(* Timer *)
WaitValve		(IN:=  bValveTime, PT:=STRING_TO_TIME(CONCAT(tempTime, 'ms')), Q=>, ET=>); 		(*Timer*)		(* For waiting for Valves 				*)
Wait			(IN:=  bWait			, PT:=T#200MS, Q=>, ET=>); 		(*Timer*)		(* For testing 							*)
Wait2			(IN:=  bWait2			, PT:=T#2500MS, Q=>, ET=>);		(*Timer*)		(* For waiting for stem to stand still 	*)
WaitMotorDrive	(IN:=  bDriveTime		, PT:=T#500MS, Q=>, ET=>);		(*Timer*)		(* For Homing 							*)

(* uiStepsToMove			-->	Antal pulser på tællerkort	:	24 Pulser pr mm * antal mm 										*)
uiStepsToMove := INT_TO_UINT(24 * uiDistToGrab);

FB_OPEN_CUT		(ExecuteHmi := (sToolControl = 'cut-open') OR GbOpenCut, 	ControlType := 1,	Ack := uiSignalInToolAck.02, 	OutQ => uiSignalOutTool.02);
FB_CLOSE_CUT	(ExecuteHmi := (sToolControl = 'cut-close'),	ControlType := 1,	Ack := uiSignalInToolAck.03, 	OutQ => uiSignalOutTool.03);
FB_RELEASE_CUT	(ExecuteHmi := GbReleaseCut OR FB_RELEASE_CUT.Execute,	ControlType := 1,	Ack := uiSignalInToolAck.01, 	OutQ =>);
FB_OPEN_PICK	(ExecuteHmi := (sToolControl = 'pick-open') OR GbOpenPick,	ControlType := 1,	Ack := uiSignalInToolAck.04, 	OutQ => uiSignalOutTool.04);
FB_CLOSE_PICK	(ExecuteHmi := (sToolControl = 'pick-close'),	ControlType := 1,	Ack := uiSignalInToolAck.05, 	OutQ => uiSignalOutTool.05);

FB_LOAD_CUT		(ExecuteHmi := (sToolControl = 'cut-load'),		ControlType := 5, 	Ack := uiSignalInToolAck.00,	OutQ => uiSignalOutTool.00, 	OutQ2 => qValve1, 	OutQ3 => qValve2);
FB_DELOAD_CUT	(ExecuteHmi := (sToolControl = 'cut-deload') OR GbDeloadCut,	ControlType := 2, 	Ack := uiSignalInToolAck.01,	OutQ => , 	OutQ2 =>bValve1Control);

FB_OPEN_GRIP	(ExecuteHmi := (sToolControl = 'grip-open'),	ControlType := 4,	OutQ =>,);
FB_CLOSE_GRIP	(ExecuteHmi := (sToolControl = 'grip-close'),	ControlType := 3, 	OutQ => ,);

FB_BRAKE		(ControlType := 1, Ack := NOT FB_BRAKE.Execute, 	OutQ => qValve3);

IF (FB_RELEASE_CUT.Execute AND FB_RELEASE_CUT.State = 10) OR (FB_DELOAD_CUT.State = 110) THEN
	uiSignalOutTool.01 := TRUE;
ELSE
	uiSignalOutTool.01 := FALSE;
END_IF

IF (sToolControl = 'brake-activate') THEN
	FB_BRAKE.Execute := TRUE;
ELSIF (sToolControl = 'brake-deactivate') THEN
	FB_BRAKE.Execute := FALSE;
END_IF


IF GbCloseGrip OR FB_CLOSE_GRIP.Execute OR FB_CLOSE_GRIP.ExecuteHmi THEN
	FB_OPEN_GRIP.Execute := FALSE;
	qValve4 := FB_CLOSE_GRIP.OutQ;
	testing := FALSE;
END_IF
IF GbOpenGrip OR FB_OPEN_GRIP.Execute OR FB_OPEN_GRIP.ExecuteHmi THEN
	testing := TRUE;
	FB_CLOSE_GRIP.Execute := FALSE;
	qValve4 := NOT FB_OPEN_GRIP.OutQ;
END_IF


IF bValve1Control THEN
	qValve1 := TRUE;
END_IF

IF sToolControl = 'cut-close' THEN
	GbCloseCut := TRUE;
	
ELSE 
	GbCloseCut := FALSE;
END_IF

END_PROGRAM

// ---- POUs/CONTROLs/Control.TcPOU
PROGRAM Control
VAR_INPUT
	State: INT := 0;
	NewState: INT := 0;

	InternalState: INT := 0;
	InternalNewState: INT := 0;
END_VAR

VAR
	adsTest: INT;
	(* FUNCTION BLOCKS *)

	(* REALS *)
		
	(* INTEGERS *)
	(*uiTrunkPos: 		UINT;				(* Stamme position	-->	Afstand i mm.															*)
	iBunchPosZ: 		UINT;
	iStemAngle:		INT;

	uiCutCoordX: 		UINT;
	uiCutCoordY: 		UINT;
	uiCutCoordZ: 		UINT;

	iStemPosX: 		UINT;				(* *)
	iStemPosY: 		UINT;				(* *)
	iStemPosZ: 		UINT;
	iRoll: 			INT;
	iPitch: 			UINT;
	iYaw:			INT;
	iPickAngle: 		INT;*)

	ImageRetryHeight:	INT;

	iMoved: 			INT;					(* Hvor mange gange har cut bevæget sig efter iBunchPosZ er nået *)
	iCnfgChange:		INT := 0;
	uiDeleaf: 		UINT;

	(* BOOLS *)
	bStopped: BOOL;
	bRobotFail: BOOL;

	bRetry: INT;
	bStemGrabbed: BOOL;

	cartMoved: BOOL;
	cartX: USINT;
	testbreak: BOOL;
	distCutJoint: INT;
	cutMin: INT;
	testFail: BOOL;
	break: BOOL;
END_VAR

CASE State OF

	0: (* init - Every important variables will be resat before the start of the sequence *)
		IF bStart AND uiprogNo = 6 AND State <> 2000  AND NOT bAlarmState THEN
			uiStatus := 1;
			FB_BRAKE.Execute := TRUE;

			(* Init variables *)
			bRetry := 0;
			uiCalibImgCount	:= 0;
			iMoved := 0;
			iImageZone := 0;
			gJointFound := 0;
			gResetPcCom 	:= TRUE;
			iCnfgChange := 0;
			uiDeleaf := 0;
			bPosSentToPcCom := FALSE;
			gStopped := FALSE;

			(* Before starting - Home *)
			GbHomeGripStem := TRUE;
			IF bHomeDone THEN
				bStart := FALSE;
				bHomeDone := FALSE;
				NewState := 10;
			END_IF
		END_IF

	10:	(* Set velocity - Both Cut and Pick *)
		bLog := TRUE;	// Starts logging of data in this Control sequence
	
		FB_SET_VELOCITY.Execute := TRUE;
		uiSignalOutSpeedControl := PROGRAM_DATA.usiVelocity;
		uiSignalOutControl := FB_SET_VELOCITY.OutQ;
		IF FB_SET_VELOCITY.Done THEN
			FB_SET_VELOCITY.Execute := FALSE;
			NewState := 20;
		END_IF

	20:	(* Idle - Both Cut and Pick *)
		FB_MOVE_TO_IDLE.Execute := TRUE;
		uiSignalOutControl := FB_MOVE_TO_IDLE.OutQ;
		IF FB_MOVE_TO_IDLE.Done THEN
			FB_MOVE_TO_IDLE.Execute := FALSE;
			NewState := 30;
		END_IF




		(* ------------------------------------------------------------------- Get Stem  ------------------------------------------------------------------- *)
	30:	(*  Load cutter *)
		FB_LOAD_CUT.Execute := TRUE;
		IF FB_LOAD_CUT.Done THEN
			FB_LOAD_CUT.Execute := FALSE;
			NewState := 35;
		END_IF
		
	35:
		(* Close grip - for it not to be in the images from CutCam *)
		FB_CLOSE_GRIP.Execute := TRUE;
		IF FB_CLOSE_GRIP.Done THEN
			FB_CLOSE_GRIP.Execute := FALSE;
			NewState := 40;
		END_IF

	40: (* Cam 1 Take image	-	parameters recieved from Vision = height of lowest ripe tomato and Y coord for lowest point of the stem *)

		FB_CAM_ONE_CONTROL.Execute := TRUE;
		IF FB_CAM_ONE_CONTROL.Done THEN
			FB_CAM_ONE_CONTROL.Execute := FALSE;
			IF FB_CAM_ONE_CONTROL.Fail THEN
				(* Adjust cart height  in order to retry *)
				NewState := 1000;
			ELSE
				(* uiDistToGrab 	-->		Distance from Joris Gripper to stem 			*)
				uiDistToGrab	:= FB_CAM_ONE_CONTROL.TrunkDist;
				(* iBunchPosZ	-->		Height of the lowest hanging red tomato		*)
				iBunchPosZ 	:= FB_CAM_ONE_CONTROL.BunchHeight;
				(* i StemAngle	-->		Heading direction from stem to lowest tomato	*)
				iStemAngle	:= FB_CAM_ONE_CONTROL.StemHeading;
				(* iImageZone	-->		Zone of lowest tomato						*)
				iImageZone	:= FB_CAM_ONE_CONTROL.Zone;
				usiImageLog := usiImageLog + 1;
				NewState := 45;
			END_IF
		END_IF

	45: (* Open gripper after  *)
		IF bRetry < 3 THEN
			FB_OPEN_GRIP.Execute := TRUE;
			IF FB_OPEN_GRIP.Done THEN
				bRetry := bRetry + 1;
				usiRetryLog := usiRetryLog + 1;
				FB_OPEN_GRIP.Execute := FALSE;
				NewState := 50;
			END_IF
		ELSE
			NewState := 1000;
		END_IF


	50:				(* Joris gripper retreives stem *)
		(* Grab stem and pull in *)
		IF NOT bAck THEN
			(* HMI knap der kalder GribStem *)
			GbGripStem := TRUE;
		ELSIF bAck THEN
			gResetPcCom := TRUE;
			NewState := 55;
		END_IF

	55:
		(* Check if stem is grabed *)
		IF uiToolState = 0 THEN
			(* Retry to grab the stem with a larger uiDistToGrab *)
			IF bJorisSensor THEN
				CASE bRetry OF
					0:
						// Retry 50mm further aways
						uiDistToGrab := uiDistToGrab + 50;
						NewState := 45;
						
					1:
						// Why?
						uiDistToGrab := uiDistToGrab - 50;
						NewState := 60;
						
					2:
						(* Keep trying intil the stem is grabed *)
						bRetry := 0;
						
				ELSE
					NewState := 1000;
				END_CASE
			ELSE
				bRetry := 0;
				NewState := 100;
			END_IF
		END_IF
		
	60:
		(* Move cart so that the *)
		IF FB_CAM_ONE_CONTROL.TrunkPosX > 280 THEN
			(* Move cart forward *)
			(* Move cart FB_CAM_ONE_CONTROL.TrunkPosX - 280 *)
			cartMoved := TRUE;
		ELSE
			(* Move cart backward *)
			(* Move cart 280 - FB_CAM_ONE_CONTROL.TrunkPosX *)
			cartMoved := TRUE;
		END_IF
		NewState := 70;
	
	70:
		IF cartMoved THEN
			(* Take a new photo and retry *)
			IF bRetry < 2 THEN
				cartMoved := FALSE;
				usiRetryLog := usiRetryLog + 1;
				NewState := 40;
			ELSE
				cartMoved := FALSE;
				NewState := 45;
			END_IF
		END_IF














	(* ------------------------------------------------------------------- Grab Stem  ------------------------------------------------------------------- *)
	100:		(* Robot Pick move to Image Pos *)
		
		IF (ABS(iStemAngle) >= 90) THEN
			IF iStemAngle < 0 THEN
				gTomatoHeading := INT_TO_BYTE(270 - ABS(iStemAngle));
			ELSE
				gTomatoHeading := INT_TO_BYTE(ABS(iStemAngle) - 90);
			END_IF
		ELSE
			gTomatoHeading := 0;
		END_IF
		
		(*IF iStemAngle < 0 THEN
			gTomatoHeading := INT_TO_BYTE(ABS(iStemAngle));
		ELSE
			gTomatoHeading := 0;
		END_IF*)
		
		FB_PICK_TRUNK_IMAGE.Execute := TRUE;
		uiSignalOutControl := FB_PICK_TRUNK_IMAGE.OutQ;
		IF FB_PICK_TRUNK_IMAGE.Done THEN
			IF uiSignalInRobotFail.00 AND testFail THEN		// Hvad er testFail?
				NewState := 1000;
				bBackToZero := TRUE;
			ELSE
				FB_PICK_TRUNK_IMAGE.Execute := FALSE;
				gResetPcCom := TRUE;
				NewState := 110;
			END_IF
		END_IF

	110:		(* Send Robot Pick Position *)
		getPickCoords := TRUE;
		IF bPosSentToPcCom AND FB_GET_PICK_COORD.Execute = FALSE THEN
			ImageRetryHeight := stDataToVision.CoordZR2G;
			bPosSentToPcCom := FALSE;
			bGetCoordDone := FALSE;
			NewState := 120;
		END_IF

	120:		(* Cam 2 take image *)
		(* Take bottom Image *)
		(* If pick coordinates are recieved, take an image *)
		IF stDataToVision.CoordXR2G <> 0 AND stDataToVision.CoordYR2G <> 0 AND stDataToVision.CoordZR2G <> 0 THEN
			FB_CAM_TWO_CONTROL.Execute := TRUE;
			IF FB_CAM_TWO_CONTROL.Done THEN
				(* If the positions was unacceptable  - Prepare to take a new picture from 50 mm further up *)
				IF FB_CAM_TWO_CONTROL.Fail THEN
					(* Send new pos to Robots *)
					GviX	:= stDataToVision.CoordXR2G / 10;
					GviY 	:= stDataToVision.CoordYR2G / 10;
					GviZ 	:= (stDataToVision.CoordZR2G / 10) + 50;

					(* GsendCoord			-->	Starter SendCoordinates sekvensen							-	Sender koordinater til robotterne 		*)
					(* uiSignalOutShared.06	-->	Bekræftelse på at koordinaterne er sendt til udgangene i box 10	-	Acknowledge fra SendCoordinates	*)
					GsendCoord := TRUE;
					IF uiSignalOutShared.06 THEN
						(* Send_pos	-->	Kommando der fortæller robot cut at nogle nye positioner er sendt *)
						uiSignalOutControl := Send_pos;
					END_IF
					IF uiSignalInAck = Send_pos THEN
						FB_CAM_TWO_CONTROL.Execute := FALSE;
						uiSignalOutControl := 0;
						uiCalibImgCount := uiCalibImgCount + 1;
						usiImageLog := usiImageLog + 1;
						NewState := 130;
					END_IF
				ELSE
					(* If positions are acceptable and stem is found, Send the posiotions to the robots *)
					FB_CAM_TWO_CONTROL.Execute := FALSE;
					IF stDataFromVision.gStemFound = 1 THEN
						IF (FB_CAM_TWO_CONTROL.X < 400) AND (FB_CAM_TWO_CONTROL.Y < 450) AND (FB_CAM_TWO_CONTROL.Z < 1000) and (FB_CAM_TWO_CONTROL.X > 0) AND (FB_CAM_TWO_CONTROL.Y > 150) AND (FB_CAM_TWO_CONTROL.Z > 200) THEN
							GviX	:= FB_CAM_TWO_CONTROL.X;
							GviY 	:= FB_CAM_TWO_CONTROL.Y;
							//Hvis joint fundet, tag fat 10cm længere nede.
							IF stDataFromVision.gJointFound = 1 THEN
								GviZ 	:= FB_CAM_TWO_CONTROL.Z - 100;
							ELSE
								GviZ 	:= FB_CAM_TWO_CONTROL.Z;
							END_IF
							//Tjek om klasen hænger i vejen for CutTool. Hvis ja, tag fat længere nede.
							IF iStemAngle < -75 AND iStemAngle > -105 AND FB_CAM_TWO_CONTROL.Z > iBunchPosZ THEN
								GviZ := iBunchPosZ;
							END_IF
							IF GviZ < 200 THEN
								GviZ := 200;
							END_IF
							GviA 	:= FB_CAM_TWO_CONTROL.RotZ0;
							GviE 	:= FB_CAM_TWO_CONTROL.RotY;
							GviR 	:= FB_CAM_TWO_CONTROL.RotZ1;
	
							GviX2 	:= FB_CAM_TWO_CONTROL.X;
							GviY2 	:= (FB_CAM_TWO_CONTROL.Y + FB_CAM_TWO_CONTROL.Y + FB_CAM_ONE_CONTROL.Y)/3;
							GviZ2	:= GviZ;
							(*GviZ2 	:= FB_CAM_ONE_CONTROL.Z + 50;*)
	
							iImageZone	:= FB_CAM_ONE_CONTROL.Zone;
							usiImageLog := usiImageLog + 1;
							NewState := 150;
						END_IF
					(* IF the stem cannot be found, retry grabbing the stem with Joris gripper *)
					ELSE
						IF bRetry = 0 THEN
							bRetry := 1;
							usiRetryLog := usiRetryLog + 1;
							gResetPcCom := TRUE;
							NewState := 110;
						ELSE
							gResetPcCom := TRUE;
							bRetry := 1000;
							bBackToZero := TRUE;
						END_IF
					END_IF
				END_IF
			END_IF
		END_IF


	130:
		IF uiSignalInAck = 0 THEN
			IF bRetry = 0 THEN
				bRetry := bRetry + 1;
				usiRetryLog := usiRetryLog + 1;
				NewState := 100;
			ELSE
				bRetry := 1000;
				bBackToZero := TRUE;
			END_IF
		END_IF

	150:		(* Send Pos to Robot *)

		(* GsendCoord			-->	Starter SendCoordinates sekvensen							-	Sender koordinater til robotterne 		*)
		(* uiSignalOutShared.06	-->	Bekræftelse på at koordinaterne er sendt til udgangene i box 10	-	Acknowledge fra SendCoordinates	*)
		GsendCoord := TRUE;
		IF uiSignalOutShared.06 THEN
			(* Send_pos	-->	Kommando der fortæller robot cut at nogle nye positioner er sendt *)
			uiSignalOutControl := Send_two_pos;
		END_IF

		IF uiSignalInAck = Send_two_pos THEN
			uiSignalOutControl := 0;
			uiCalibImgCount := uiCalibImgCount + 1;
			NewState := 155;
		END_IF


	155:
		IF uiSignalInAck = 0 THEN
			NewState := 160;
		END_IF

	160:		(* Grab the stem + Move to image pos *)
		FB_IMAGE_GRAB.Execute := TRUE;
		uiSignalOutControl := FB_IMAGE_GRAB.OutQ;

		IF FB_IMAGE_GRAB.Done THEN
			IF uiSignalInRobotFail.00 AND testFail THEN
				NewState := 1000;
				bBackToZero := TRUE;
			ELSE
				FB_IMAGE_GRAB.Execute := FALSE;
				NewState := 200;
			END_IF
		END_IF









	(* ------------------------------------------------------------------- "WHAT IF" FIXES  ------------------------------------------------------------------- *)
	200:
		IF NOT bRobotFail THEN
			bRetry := 0;
			gResetPcCom := TRUE;
			NewState := 250;
		ELSE
			(* Retries:																						*)
			(* Open and close cone								-	To check if it was a misreading from sensor 	*)
			(* Move to pos 50mm above normal image pos, then retry												*)
			IF bRetry  < 2 THEN
				bRetry := bRetry + 1;
				usiRetryLog := usiRetryLog + 1;
				(*uiCalibImgCount := 0;*)
				GviZ2 := stDataToVision.CoordZR2G/10 + 100;
				NewState := 220;
			ELSE
				bBackToZero := TRUE;
			END_IF
		END_IF


	220:
		(* GsendCoord			-->	Starter SendCoordinates sekvensen							-	Sender koordinater til robotterne 		*)
		(* uiSignalOutShared.06	-->	Bekræftelse på at koordinaterne er sendt til udgangene i box 10	-	Acknowledge fra SendCoordinates	*)
		GsendCoord := TRUE;
		IF uiSignalOutShared.06 THEN
			(* Send_pos	-->	Kommando der fortæller robot cut at nogle nye positioner er sendt *)
			uiSignalOutControl := Send_two_pos;
		END_IF

		IF uiSignalInAck = Send_two_pos THEN
			uiSignalOutControl := 0;
			NewState := 225;
		END_IF

	225:
		IF uiSignalInAck = 0 THEN
			gResetPcCom := TRUE;
			NewState := 230;
		END_IF


	230:		(* Retry Grab Stem *)
		FB_RETRY_GRAB_STEM.Execute := TRUE;
		uiSignalOutControl := FB_RETRY_GRAB_STEM.OutQ;
		IF FB_RETRY_GRAB_STEM.Done THEN
			FB_RETRY_GRAB_STEM.Execute := FALSE;
			gResetPcCom := TRUE;
			NewState := 110;
		END_IF










	(* ------------------------------------------------------------------- Move On Stem  ------------------------------------------------------------------- *)
	250:		(* Send Robot Pick Position *)
		getPickCoords := TRUE;
		IF bPosSentToPcCom AND FB_GET_PICK_COORD.Execute = FALSE THEN
			ImageRetryHeight := stDataToVision.CoordZR2G;
			bPosSentToPcCom := FALSE;
			bGetCoordDone := FALSE;
			NewState := 260;
		END_IF

	260:
		IF stDataToVision.CoordXR2G <> 0 AND stDataToVision.CoordYR2G <> 0 AND stDataToVision.CoordZR2G <> 0 THEN
			FB_CAM_TWO_CONTROL.Execute := TRUE;
			IF FB_CAM_TWO_CONTROL.Done THEN
				FB_CAM_TWO_CONTROL.Execute := FALSE;
				(* Check if the stem is found *)
				IF FB_CAM_TWO_CONTROL.StemFound = 1 THEN
					IF FB_CAM_TWO_CONTROL.X > 350 OR FB_CAM_TWO_CONTROL.X < 200 OR FB_CAM_TWO_CONTROL.Y > 350 OR FB_CAM_TWO_CONTROL.Y < 200 THEN
						GviX := 320;
						GviY := 320;
						IF (stDataFromVision.ResultPar3 < iBunchPosZ) THEN
							GviZ := FB_CAM_TWO_CONTROL.Z;
						ELSE
							GviZ := iBunchPosZ;
						END_IF
						GviA := 0;
						GviE := 0;
						GviR := 40;
					ELSE
						GviX := (FB_CAM_TWO_CONTROL.X + 320) / 2;
						GviY := (FB_CAM_TWO_CONTROL.Y + 320) / 2;
						IF (stDataFromVision.ResultPar3 < iBunchPosZ) THEN
							GviZ := FB_CAM_TWO_CONTROL.Z;
						ELSE
							GviZ := iBunchPosZ;
						END_IF
						GviA := 0;
						GviE := 0;
						GviR := 40;
					END_IF
					(*IF FB_CAM_TWO_CONTROL.JointFound = 1 THEN
						GviPick := FB_CAM_TWO_CONTROL.PickAngle;
						iImageZone := FB_CAM_TWO_CONTROL.Zone;
						gResetPcCom := TRUE;
						NewState := 310;
					ELSE*)
					usiImageLog := usiImageLog + 1;
						gResetPcCom := TRUE;
						NewState := 270;
					(*END_IF*)
				ELSE
					usiImageLog := usiImageLog + 1;
					gResetPcCom := TRUE;
					NewState := 345;
				END_IF
			END_IF
		END_IF

	270:
		(* Send pos to Robots *)
		(* GsendCoord			-->	Starter SendCoordinates sekvensen							-	Sender koordinater til robotterne 		*)
		(* uiSignalOutShared.06	-->	Bekræftelse på at koordinaterne er sendt til udgangene i box 10	-	Acknowledge fra SendCoordinates	*)
		GsendCoord := TRUE;
		IF uiSignalOutShared.06 THEN
			(* Send_pos	-->	Kommando der fortæller robot cut at nogle nye positioner er sendt *)
			uiSignalOutControl := Send_pos;
		END_IF
		IF uiSignalInAck = Send_pos THEN
			uiSignalOutControl := 0;
			uiCalibImgCount := uiCalibImgCount + 1;
			NewState := 275;
		END_IF

	275:
		IF uiSignalInAck = 0 THEN
			NewState := 280;
		END_IF

	280:		(* CO-MOVE up the stem *)
		FB_COMOVE_IMAGE.Execute := TRUE;
		uiSignalOutControl := FB_COMOVE_IMAGE.OutQ;
		IF FB_COMOVE_IMAGE.Done THEN
			IF uiSignalInRobotFail.00 AND testFail THEN
				NewState := 1000;
				bBackToZero := TRUE;
			ELSE
				FB_COMOVE_IMAGE.Execute := FALSE;
				IF bRobotFail THEN
					NewState := 3000;
				ELSE
					NewState := 290;
				END_IF
			END_IF
		END_IF

	290:
		(* Send Pick coordinate *)
		(* Send Pick pos to PcCom for next image *)
		getPickCoords := TRUE;
		IF bPosSentToPcCom AND FB_GET_PICK_COORD.Execute = FALSE THEN
			bPosSentToPcCom := FALSE;
			NewState := 300;
		END_IF











	(* ------------------------------------------------------------------- Find Joint  ------------------------------------------------------------------- *)
	300:		(* Take a picture *)
		IF stDataToVision.CoordXR2G <> 0 AND stDataToVision.CoordYR2G <> 0 AND stDataToVision.CoordZR2G <> 0 THEN
			FB_CAM_TWO_CONTROL.Execute := TRUE;
			IF FB_CAM_TWO_CONTROL.Done THEN
				IF FB_CAM_TWO_CONTROL.StemFound = 1 THEN
					IF FB_GET_CUT_COORD.Execute = FALSE THEN
						IF FB_CAM_TWO_CONTROL.Zone <> 0 THEN
							iImageZone := FB_CAM_TWO_CONTROL.Zone;
						END_IF
						IF distCutJoint = 0 THEN
							(* Get Cut coord *)
							gResetPcCom := TRUE;
							getCutCoords := TRUE;
							bGetCutCoordDone:= FALSE;
							cutMin := 15;	(* Max lenght from top of cut head to joint*)
						END_IF
						IF FB_CAM_TWO_CONTROL.X > 350 OR FB_CAM_TWO_CONTROL.X < 200 OR FB_CAM_TWO_CONTROL.Y > 350 OR FB_CAM_TWO_CONTROL.Y < 200 THEN
							usiImageLog := usiImageLog + 1;
							NewState := 302;							
						ELSE
							usiImageLog := usiImageLog + 1;
							NewState := 303;
						END_IF
					END_IF
				ELSE
					FB_CAM_TWO_CONTROL.Execute := FALSE;
					gResetPcCom := TRUE;
					usiImageLog := usiImageLog + 1;
					NewState := 345;
				END_IF
			END_IF
		END_IF
		
	302:
		IF bGetCutCoordDone THEN
			bGetCutCoordDone:= FALSE;
			distCutJoint := stDataFromVision.ResultPar3 - (currentRobotZ / 10);
		
			IF distCutJoint <> 0 OR ((stDataFromVision.ResultPar3 = (currentRobotZ/10)) AND (currentRobotZ <> 0)) THEN
				IF FB_CAM_TWO_CONTROL.JointFound = 1 AND distCutJoint <= cutMin THEN
					GviPick := FB_CAM_TWO_CONTROL.PickAngle;

					getCutCoords := TRUE;
					IF FB_CAM_TWO_CONTROL.TrussFound = 1 THEN
						iCnfgChange := 0;
					END_IF
					IF bPosSentToPcCom AND FB_GET_CUT_COORD.Execute = FALSE THEN
						bPosSentToPcCom := FALSE;
						FB_CAM_TWO_CONTROL.Execute := FALSE;
						gResetPcCom := TRUE;
						NewState := 305;
					END_IF
				ELSE
					GviX := 320;
					GviY := 320;
					GviZ := FB_CAM_TWO_CONTROL.Z;

					GviA 	:= 0;
					GviE 	:= 0;
					GviR 	:= 40;

					FB_CAM_TWO_CONTROL.Execute := FALSE;
					gResetPcCom := TRUE;
					iCnfgChange := 0;
					NewState := 310;
				END_IF
			END_IF
		END_IF
		
	303:
		IF bGetCutCoordDone THEN
			bGetCutCoordDone:= FALSE;
			distCutJoint := stDataFromVision.ResultPar3 - (currentRobotZ / 10);
		
			IF distCutJoint <> 0 OR ((stDataFromVision.ResultPar3 = (currentRobotZ/10)) AND (currentRobotZ <> 0)) THEN
				IF FB_CAM_TWO_CONTROL.JointFound = 1 AND distCutJoint <= cutMin THEN
					GviPick := FB_CAM_TWO_CONTROL.PickAngle;
					IF FB_CAM_TWO_CONTROL.TrussFound = 1 THEN
						iCnfgChange := 0;
					END_IF
					IF bPosSentToPcCom THEN
						bPosSentToPcCom := FALSE;
						FB_CAM_TWO_CONTROL.Execute := FALSE;
						NewState := 305;
					END_IF
				ELSIF distCutJoint > cutMin THEN
					IF FB_CAM_TWO_CONTROL.JointFound = 1 THEN
						GviZ := FB_CAM_TWO_CONTROL.Z - 10;
						iCnfgChange := 0;
					ELSE
						GviZ := FB_CAM_TWO_CONTROL.Z;
					END_IF
					GviX := (FB_CAM_TWO_CONTROL.X + 320) / 2;
					GviY := (FB_CAM_TWO_CONTROL.Y + 320) / 2;
					GviA 	:= 0;
					GviE 	:= 0;
					GviR 	:= 40;

					FB_CAM_TWO_CONTROL.Execute := FALSE;
					gResetPcCom := TRUE;
					NewState := 310;
				ELSE
					bBackToZero := TRUE;
				END_IF
			END_IF
		END_IF

	305:
		IF uiSignalInAck = 0 THEN
			GviX	:= stDataToVision.CoordXR1G / 10;
			GviY	:= stDataToVision.CoordYR1G / 10;
			GviZ	:= stDataToVision.CoordZR1G / 10;
			gResetPcCom := TRUE;
			NewState := 310;
		END_IF

	310:		(* Send pos *)
		(* GsendCoord			-->	Starter SendCoordinates sekvensen							-	Sender koordinater til robotterne 		*)
		(* uiSignalOutShared.06	-->	Bekræftelse på at koordinaterne er sendt til udgangene i box 10	-	Acknowledge fra SendCoordinates	*)
		IF (FB_CAM_TWO_CONTROL.TomatoFound = 1) AND (FB_CAM_TWO_CONTROL.JointFound <> 1) THEN
			NewState := 315;
		ELSE
			GsendCoord := TRUE;
			IF uiSignalOutShared.06 THEN
				(* Send_pos	-->	Kommando der fortæller robot cut at nogle nye positioner er sendt *)
				uiSignalOutControl := Send_pos;
			END_IF
			IF uiSignalInAck = Send_pos THEN
				uiSignalOutControl := 0;
				(*uiCalibImgCount := uiCalibImgCount + 1;*)
				NewState := 315;
			END_IF
		END_IF

	315:
		IF uiSignalInAck = 0 THEN
			IF FB_CAM_TWO_CONTROL.JointFound = 1 AND stDataFromVision.ResultPar3 > iBunchPosZ AND (currentRobotZ/10) > iBunchPosZ AND distCutJoint < cutMin THEN
				NewState := 345;
			ELSIF (FB_CAM_TWO_CONTROL.TomatoFound = 1) AND (FB_CAM_TWO_CONTROL.JointFound <> 1) AND (stDataFromVision.ResultPar3 > iBunchPosZ) AND iCnfgChange < 6 THEN
				iCnfgChange := iCnfgChange + 1;
				usiImageRetry := usiImageRetry + 1;
				IF uiCalibImgCount < 50 THEN
					uiCalibImgCount := 50;
				END_IF
				IF uiCalibImgCount >= 50 AND uiCalibImgCount <= 200 THEN
					NewState := 350;
				ELSIF uiCalibImgCount = 250 THEN
					NewState := 450;
				END_IF
			ELSE
				NewState := 320;
			END_IF
		END_IF
	320:
		FB_COMOVE_IMAGE.Execute := TRUE;
		uiSignalOutControl := FB_COMOVE_IMAGE.OutQ;
		IF FB_COMOVE_IMAGE.Done THEN
			FB_COMOVE_IMAGE.Execute := FALSE;
			IF uiSignalInRobotFail.00 AND testFail THEN
				NewState := 1000;
				bBackToZero := TRUE;
			ELSE
				IF bRobotFail THEN
					NewState := 3000;
				ELSE
					IF FB_CAM_TWO_CONTROL.JointFound = 1 AND distCutJoint > cutMin AND stDataFromVision.ResultPar3 < iBunchPosZ AND FB_CAM_TWO_CONTROL.TrussFound = 0 THEN
						NewState := 325;
					ELSE
						NewState := 330;
					END_IF
				END_IF
			END_IF
		END_IF

	325:
		FB_RELEASE_CUT.Execute := TRUE;
		IF FB_RELEASE_CUT.Done THEN
			usiStickoutCutLog := usiStickoutCutLog + 1;
			FB_RELEASE_CUT.Execute := FALSE;
			NewState := 327;
		END_IF

	327:
		FB_LOAD_CUT.Execute := TRUE;
		IF FB_LOAD_CUT.Done THEN
			FB_LOAD_CUT.Execute := FALSE;
			NewState := 330;
		END_IF


	330: 		(* Send Pick coordinate *)
		(* Send Pick pos to PcCom for next image *)
		getPickCoords := TRUE;
		IF bPosSentToPcCom AND FB_GET_PICK_COORD.Execute = FALSE THEN
			bPosSentToPcCom := FALSE;
			NewState := 345;
		END_IF

	345:
		IF uiSignalInAck = 0 THEN
			IF stDataFromVision.gJointFound = 1 (*AND stDataFromVision.ResultPar3 > iBunchPosZ*) AND FB_CAM_TWO_CONTROL.StemFound = 1 AND distCutJoint < cutMin AND FB_CAM_TWO_CONTROL.TrussFound = 1 (*AND FB_CAM_TWO_CONTROL.TomatoFound = 1*) THEN
				(* Grabbing sequence *)
				gResetPcCom := TRUE;
				IF uimodeNo <= 1 THEN
					NewState := 400;
				ELSE
					NewState := 420;
				END_IF
			ELSIF stDataFromVision.gJointFound = 1 AND stDataFromVision.ResultPar3 > iBunchPosZ AND FB_CAM_TWO_CONTROL.StemFound = 1 AND distCutJoint < cutMin AND FB_CAM_TWO_CONTROL.TrussFound = 0 (*AND FB_CAM_TWO_CONTROL.TomatoFound = 1*) THEN
				iCnfgChange := iCnfgChange + 1;
				usiImageRetry := usiImageRetry + 1;
				NewState := 350;
			ELSIF stDataFromVision.gStemFound = 1 AND iMoved < 2 THEN
				(* Move further Along stem *)
				NewState := 360;
			ELSIF stDataFromVision.gStemFound = 0 OR iMoved >= 2 THEN
				(* Change configuration *)
				iCnfgChange := iCnfgChange + 1;
				usiImageRetry := usiImageRetry + 1;
				IF uiCalibImgCount >= 50 AND uiCalibImgCount <= 200 THEN
					NewState := 350;
				ELSIF uiCalibImgCount = 250 THEN
					NewState := 450;
				END_IF
				gResetPcCom := TRUE;
				NewState := 350;
			ELSIF stDataFromVision.gJointFound = 255 THEN 	(* If timeout *)
				bBackToZero := TRUE;
			END_IF
		END_IF
		distCutJoint := 0;

	(* ------------------------------------------ Change configuration ------------------------------------------ *)
	350:
		IF iCnfgChange <= 5 THEN
			uiCalibImgCount := INT_TO_BYTE(iCnfgChange * 50);
		ELSE
			bBackToZero := TRUE;
		END_IF
		(* Robot Pick to image pos *)
		FB_PICK_TRUNK_IMAGE.Execute := TRUE;
		uiSignalOutControl := FB_PICK_TRUNK_IMAGE.OutQ;
		IF FB_PICK_TRUNK_IMAGE.Done THEN
			IF uiSignalInRobotFail.00 AND testFail THEN
				NewState := 1000;
				bBackToZero := TRUE;
			ELSE
				FB_PICK_TRUNK_IMAGE.Execute := FALSE;
				NewState := 360;
			END_IF
		END_IF

	360:		(* Send Pick coordinate *)
		(* Send Pick pos to PcCom for next image *)
		getPickCoords := TRUE;
		IF bPosSentToPcCom THEN
			bPosSentToPcCom := FALSE;
			NewState := 300;
		END_IF


	(* ------------------------------------------ Grab tomatoes ------------------------------------------ *)
	400:		(* Robot Pick grab *)
		FB_PICK_GRAB.Execute := TRUE;
		uiSignalOutControl := FB_PICK_GRAB.OutQ;
		IF FB_PICK_GRAB.Done THEN
			FB_PICK_GRAB.Execute := FALSE;
			IF uiSignalInRobotFail.00 AND testFail THEN
				NewState := 2000;
				(*NewState := 1000;
				bBackToZero := TRUE;*)
			ELSE
				IF NOT bRobotFail THEN
					bRetry := 0;
					NewState := 420;
				ELSE
					IF bRetry = 0 THEN
						(* Take a new picture *)
						bRetry := 1;
						usiRetryLog := usiRetryLog + 1;
						NewState := 350;
					ELSE
						bBackToZero := TRUE;
					END_IF
				END_IF
			END_IF
		END_IF

	420:		(* Cut *)
		FB_RELEASE_CUT.Execute := TRUE;
		IF FB_RELEASE_CUT.Done THEN
			FB_RELEASE_CUT.Execute := FALSE;
			NewState := 425;
		END_IF

	425:		(* Load Cut *)
		FB_LOAD_CUT.Execute := TRUE;
		IF FB_LOAD_CUT.Done THEN
			FB_LOAD_CUT.Execute := FALSE;
			IF uimodeNo <= 1 THEN
				NewState := 430;
			ELSE
				NewState := 500;
			END_IF
		END_IF

	430:		(* Move from pick *)
		FB_PICK_MOVE_FROM_PICK.Execute := TRUE;
		uiSignalOutControl := FB_PICK_MOVE_FROM_PICK.OutQ;
		IF FB_PICK_MOVE_FROM_PICK.Done THEN
			FB_PICK_MOVE_FROM_PICK.Execute := FALSE;
			IF uiSignalInRobotFail.00 AND testFail THEN
				NewState := 1000;
				bBackToZero := TRUE;
			ELSE
				iMoved := 1;
				IF uimodeNo = 1 THEN
					NewState := 500;
				ELSE
					NewState := 540;
				END_IF
			END_IF
		END_IF
	
	450:
		bBackToZero := TRUE;

	(* --------------------------------- DELEAFING ------------------------------------ *)
	500:		(* Image of LEAFS *)
		uiCalibImgCount := INT_TO_BYTE(iMoved * 50);
		FB_PICK_DELEAF_PROGRAM.Execute := TRUE;
		uiSignalOutControl := FB_PICK_DELEAF_PROGRAM.OutQ;
		IF FB_PICK_DELEAF_PROGRAM.Done THEN
			iMoved := iMoved + 1;
			FB_PICK_DELEAF_PROGRAM.Execute := FALSE;
			NewState := 520;
		END_IF

	520:		(* Send Pick coordinate *)
		getPickCoords := TRUE;
		IF bPosSentToPcCom AND FB_GET_PICK_COORD.Execute = FALSE THEN
			bPosSentToPcCom := FALSE;
			NewState := 530;
		END_IF

	530:
		IF stDataToVision.CoordXR2G <> 0 AND stDataToVision.CoordYR2G <> 0 AND stDataToVision.CoordZR2G <> 0 THEN
			FB_CAM_TWO_CONTROL.Execute := TRUE;
			IF FB_CAM_TWO_CONTROL.Done THEN
				IF FB_CAM_TWO_CONTROL.StemFound = 1 THEN
					IF FB_CAM_TWO_CONTROL.X > 500 OR FB_CAM_TWO_CONTROL.X < 200 OR FB_CAM_TWO_CONTROL.Y > 425 OR FB_CAM_TWO_CONTROL.Y < 200 THEN
						FB_CAM_TWO_CONTROL.Execute := FALSE;
						NewState := 1000;
					ELSE
						IF FB_CAM_TWO_CONTROL.JointFound = 1 THEN
							GviX := FB_CAM_TWO_CONTROL.X;
							GviY := FB_CAM_TWO_CONTROL.Y;
							GviZ := FB_CAM_TWO_CONTROL.Z;
							GviA := 0;
							GviE := 0;
							GviR := 40;
							GviPick := FB_CAM_TWO_CONTROL.PickAngle;
							iImageZone := FB_CAM_TWO_CONTROL.Zone;
							gJointFound := FB_CAM_TWO_CONTROL.JointFound;
							FB_CAM_TWO_CONTROL.Execute := FALSE;
							gResetPcCom := TRUE;
							NewState := 540;
						ELSE
							gJointFound := FB_CAM_TWO_CONTROL.JointFound;
							FB_CAM_TWO_CONTROL.Execute := FALSE;
							gResetPcCom := TRUE;
							NewState := 500;
						END_IF
					END_IF
				ELSIF iMoved > 3 THEN
					gJointFound := FB_CAM_TWO_CONTROL.JointFound;
					FB_CAM_TWO_CONTROL.Execute := FALSE;
					gResetPcCom := TRUE;
					NewState := 540;
				ELSE
					FB_CAM_TWO_CONTROL.Execute := FALSE;
					gResetPcCom := TRUE;
					NewState := 500;
				END_IF
			END_IF
		END_IF

	540:		(* Send pos *)
		FB_PLACE.Execute := TRUE;
		IF FB_PLACE.Done THEN
			GviX2 := FB_PLACE.X;
			GviY2 := FB_PLACE.Y;
			GviZ2 := FB_PLACE.Z;
			(* GsendCoord			-->	Starter SendCoordinates sekvensen							-	Sender koordinater til robotterne 		*)
			(* uiSignalOutShared.06	-->	Bekræftelse på at koordinaterne er sendt til udgangene i box 10	-	Acknowledge fra SendCoordinates	*)
			GsendCoord := TRUE;
			IF uiSignalOutShared.06 THEN
				(* Send_pos	-->	Kommando der fortæller robot cut at nogle nye positioner er sendt *)
				uiSignalOutControl := Send_two_pos;
			END_IF
			IF uiSignalInAck = Send_two_pos THEN
				uiSignalOutControl := 0;
				uiCalibImgCount := uiCalibImgCount + 1;
				FB_PLACE.Execute := FALSE;
				NewState := 545;
			END_IF
		END_IF

	545:
		IF uiSignalInAck = 0 THEN
			NewState := 550;
		END_IF

	550:
		IF uimodeNo = 0 THEN
			FB_PLACE_DELEAF.Execute := TRUE;
			uiSignalOutControl := FB_PLACE_DELEAF.OutQ;
			IF FB_PLACE_DELEAF.Done THEN
				FB_PLACE_DELEAF.Execute := FALSE;
				NewState := 580;
			END_IF
		ELSIF uimodeNo = 1 THEN
			FB_PICK_PLACE.Execute := TRUE;
			uiSignalOutControl := FB_PICK_PLACE.OutQ;
			IF FB_PICK_PLACE.Done THEN
				FB_PICK_PLACE.Execute := FALSE;
				NewState := 600;
			END_IF
		ELSE
			FB_PICK_DELEAF_PROGRAM.Execute := TRUE;
			uiSignalOutControl := FB_PICK_DELEAF_PROGRAM.OutQ;
			IF FB_PICK_DELEAF_PROGRAM.Done THEN
				FB_PICK_DELEAF_PROGRAM.Execute := FALSE;
				NewState := 580;
			END_IF
		END_IF


	580:		(* Load Cut *)
		FB_LOAD_CUT.Execute := TRUE;
		IF FB_LOAD_CUT.Done THEN
			FB_LOAD_CUT.Execute := FALSE;
			NewState := 585;
		END_IF

	585:
		IF uiDeleaf < 0 THEN
			uiDeleaf := uiDeleaf + 1;
			NewState := 500;
		ELSE
			uiDeleaf := 0;
			NewState := 600;
		END_IF

	600:		(*Open Cut*)
		FB_OPEN_CUT.Execute := TRUE;
		IF FB_OPEN_CUT.Done THEN
			FB_OPEN_CUT.Execute := FALSE;
			NewState := 610;
		END_IF

	610:		(*Move cut away from stem*)
		FB_CUT_FROM_STEM.Execute := TRUE;
		uiSignalOutControl := FB_CUT_FROM_STEM.OutQ;
		IF FB_CUT_FROM_STEM.Done THEN
			FB_CUT_FROM_STEM.Execute := FALSE;
			NewState := 620;
		END_IF


	620:		(* GbReleaseStem *)
		(* Grab stem and pull in *)
		IF NOT bAck THEN
			(* HMI knap der kalder GribStem *)
			GbReleaseStem := TRUE;
		ELSIF bAck THEN
			NewState := 630;
		END_IF

	630:		(* Move to idle *)
		FB_MOVE_TO_IDLE.Execute := TRUE;
		uiSignalOutControl := FB_MOVE_TO_IDLE.OutQ;
		IF FB_MOVE_TO_IDLE.Done THEN
			IF uiSignalInRobotFail.00 AND testFail THEN
				NewState := 1000;
				bBackToZero := TRUE;
			ELSE
				FB_MOVE_TO_IDLE.Execute := FALSE;
				uiStatus := 0;
				NewState := 640;
			END_IF
		END_IF

	640:		(* Deload *)

		FB_DELOAD_CUT.Execute := TRUE;
		IF FB_DELOAD_CUT.Done THEN
			FB_DELOAD_CUT.Execute := FALSE;
			NewState := 650;
		END_IF

	650:
		FB_CLOSE_GRIP.Execute := TRUE;
		IF FB_CLOSE_GRIP.Done THEN
			bLogSucces := 1;
			FB_CLOSE_GRIP.Execute := FALSE;
			FB_BRAKE.Execute := FALSE;
			gStopped := TRUE;
			NewState := 0;
		END_IF



	1000:	(* Reset *)

		uiSignalOutControl  := 0;		(* Stop sequences on ROBOTS *)

		(* Reset timers *)
		bRetry := 0;
		stDataToVision.ResultRead := 1;
		gResetPcCom := TRUE;
		iCnfgChange := 1;
		uiCalibImgCount := 0;
		uiDeleaf := 0;
		InternalNewState := 0;
		NewState := 0;

	2000:
		bStopped := TRUE;


	(* ----------------------------- FAILED WHEN MOVING ON STEM ----------------------------- *)
	3000:		(* First figure out if cut is under the lowest tomato *)
		(* Get Cut coord *)
		getCutCoords := TRUE;
		IF bPosSentToPcCom AND FB_GET_CUT_COORD.Execute = FALSE THEN
			bPosSentToPcCom := FALSE;
			gResetPcCom := TRUE;
			NewState := 3005;
		END_IF

	3005:
		IF uiSignalInAck = 0 THEN
			uiCutCoordX	:= stDataToVision.CoordXR1G / 10;
			uiCutCoordY	:= stDataToVision.CoordYR1G / 10;
			uiCutCoordZ	:= stDataToVision.CoordZR1G / 10;

			NewState := 3010;
		END_IF

	3010:

		IF uiCutCoordZ > iBunchPosZ THEN
			(* Then cut must have reached the joint*)
			NewState := 330;

		ELSE
			(* It must be a too big of a stick-out *)
			FB_RELEASE_CUT.Execute := TRUE;
			IF FB_RELEASE_CUT.Done THEN
				FB_RELEASE_CUT.Execute := FALSE;
				NewState := 3020;
			END_IF
		END_IF

	3020:
		FB_LOAD_CUT.Execute := TRUE;
		IF FB_LOAD_CUT.Done THEN
			FB_LOAD_CUT.Execute := FALSE;
			NewState := 320;
		END_IF



END_CASE

IF State <> 2000 THEN
	bStopped := FALSE;
END_IF

bRobotFail := uiSignalIn2.07;

FB_PLACE(Offset := 140,		Box_length := uiBoxLength, 		Box_width := uiBoxWidth,	Box_height := uiBoxHeight,		Stem_length := 200,	Mode := uiPackingModeNo);

END_PROGRAM

// ---- POUs/CONTROLs/ControlAuto.TcPOU
PROGRAM ControlAuto
VAR_INPUT
	State: INT := 0;
	NewState: INT := 0;
END_VAR

VAR
	(* FUNCTION BLOCKS *)
	FB_PLACE: PlaceCoordinates;

	(* REALS *)

	(* INTEGERS *)
	(*uiTrunkPos: 		UINT;				(* Stamme position	-->	Afstand i mm.															*)
	iBunchPosZ: 		UINT;
	iStemAngle:		INT;

	iStemPosX: 		UINT;				(* *)
	iStemPosY: 		UINT;				(* *)
	iStemPosZ: 		UINT;
	iRoll: 			INT;
	iPitch: 			UINT;
	iYaw:			INT;
	iPickAngle: 		INT;*)

	iMoved: 			INT;					(* Hvor mange gange har cut bevæget sig efter iBundPosZ er nået *)
	iCnfgChange:		INT := 0;
	uiDeleaf: 		UINT;

	(* BOOLS *)
	bStopped: BOOL;

END_VAR

CASE State OF

	0:		(* init	-	Every important variables will be resat before the start of the sequence *)
		IF bStart AND uiprogNo = 4 AND State <> 2000  AND NOT bAlarmState THEN
			uiStatus := 1;

			(* Init variables *)
			uiCalibImgCount	:= 0;
			iMoved := 0;
			iImageZone := 0;
			gJointFound := 0;
			gResetPcCom 	:= TRUE;
			iCnfgChange := 0;
			uiDeleaf := 0;
			bPosSentToPcCom := FALSE;

			(* Before starting - Home *)
			GbHomeGripStem := TRUE;
			IF bHomeDone THEN
				bStart := FALSE;
				bHomeDone := FALSE;
				NewState := 10;
			END_IF
		END_IF

	10:		(* Set velocity *)
		FB_SET_VELOCITY.Execute := TRUE;
		uiSignalOutSpeedControl := UINT_TO_BYTE(uiSpeedSetting);
		uiSignalOutControl := FB_SET_VELOCITY.OutQ;
		IF FB_SET_VELOCITY.Done THEN
			FB_SET_VELOCITY.Execute := FALSE;
			NewState := 20;
		END_IF

	20:		(* Idle *)
		FB_MOVE_TO_IDLE.Execute := TRUE;
		uiSignalOutControl := FB_MOVE_TO_IDLE.OutQ;
		IF FB_MOVE_TO_IDLE.Done THEN
			FB_MOVE_TO_IDLE.Execute := FALSE;
			NewState := 30;
		END_IF

	30:		(*  Load cutter *)
		FB_LOAD_CUT.Execute := TRUE;
		IF FB_LOAD_CUT.Done THEN
			FB_LOAD_CUT.Execute := FALSE;
			NewState := 40;
		END_IF

	40: 		(* Cam 1 Take image	-	parameters recieved from Vision = height of lowest ripe tomato and Y coord for lowest point of the stem *)

		FB_CAM_ONE_CONTROL.Execute := TRUE;
		IF FB_CAM_ONE_CONTROL.Done THEN
			FB_CAM_ONE_CONTROL.Execute := FALSE;

			(* uiDistToGrab 	-->		Distance from Joris Gripper to stem 			*)
			uiDistToGrab	:= FB_CAM_ONE_CONTROL.TrunkDist;
			(* iBunchPosZ	-->		Height of the lowest hanging red tomato		*)
			iBunchPosZ 	:= FB_CAM_ONE_CONTROL.BunchHeight;
			(* i StemAngle	-->		Heading direction from stem to lowest tomato	*)
			iStemAngle	:= FB_CAM_ONE_CONTROL.StemHeading;
			(* iImageZone	-->		Zone of lowest tomato						*)
			iImageZone	:= FB_CAM_ONE_CONTROL.Zone;
			NewState := 50;
		END_IF

	50:		(* Joris gripper retreives stem *)
		(* Grab stem and pull in *)
		IF NOT bAck THEN
			(* HMI knap der kalder GribStem *)
			GbGripStem := TRUE;
		ELSIF bAck THEN
			gResetPcCom := TRUE;
			NewState := 55;
		END_IF

	55:
		IF uiToolState = 0 THEN
			NewState := 100;
		END_IF

	(* ---------------------------- Grab the stem ---------------------------- *)

	100:		(* Robot Pick move to Image Pos *)
		FB_PICK_TRUNK_IMAGE.Execute := TRUE;
		uiSignalOutControl := FB_PICK_TRUNK_IMAGE.OutQ;
		IF FB_PICK_TRUNK_IMAGE.Done THEN
			FB_PICK_TRUNK_IMAGE.Execute := FALSE;
			gResetPcCom := TRUE;
			NewState := 110;
		END_IF

	110:		(* Send Robot Pick Position *)
		getPickCoords := TRUE;
		IF bPosSentToPcCom AND FB_GET_PICK_COORD.Execute = FALSE THEN
			bPosSentToPcCom := FALSE;
			bGetCoordDone := FALSE;
			NewState := 120;
		END_IF

	120:		(* Cam 2 take image *)
		(* Take bottom Image *)
		(* If pick coordinates are recieved, take an image *)
		IF stDataToVision.CoordXR2G <> 0 AND stDataToVision.CoordYR2G <> 0 AND stDataToVision.CoordZR2G <> 0 THEN
			FB_CAM_TWO_CONTROL.Execute := TRUE;
			IF FB_CAM_TWO_CONTROL.Done THEN
				FB_CAM_TWO_CONTROL.Execute := FALSE;
				(* If the positionis unacceptable, reset 		-	Else, send position *)
				IF FB_CAM_TWO_CONTROL.X > 420 OR FB_CAM_TWO_CONTROL.X < 125 OR FB_CAM_TWO_CONTROL.Y > 400 OR FB_CAM_TWO_CONTROL.Y < 125 THEN
					NewState := 1000;
				ELSE
					GviX	:= FB_CAM_TWO_CONTROL.X;
					GviY 	:= FB_CAM_TWO_CONTROL.Y;
					GviZ 	:= FB_CAM_TWO_CONTROL.Z;
					GviA 	:= FB_CAM_TWO_CONTROL.RotZ0;
					GviE 	:= FB_CAM_TWO_CONTROL.RotY;
					GviR 	:= FB_CAM_TWO_CONTROL.RotZ1;

					GviX2 	:= FB_CAM_TWO_CONTROL.X;
					GviY2 	:= (FB_CAM_TWO_CONTROL.Y + FB_CAM_TWO_CONTROL.Y + FB_CAM_ONE_CONTROL.Y)/3;
					GviZ2 	:= FB_CAM_ONE_CONTROL.Z + 50;

					iImageZone	:= FB_CAM_ONE_CONTROL.Zone;
					gResetPcCom := TRUE;
					NewState := 130;
				END_IF
			END_IF
		END_IF

	130:		(* Send Pos to Robot *)

		(* GsendCoord			-->	Starter SendCoordinates sekvensen							-	Sender koordinater til robotterne 		*)
		(* uiSignalOutShared.06	-->	Bekræftelse på at koordinaterne er sendt til udgangene i box 10	-	Acknowledge fra SendCoordinates	*)
		GsendCoord := TRUE;
		IF uiSignalOutShared.06 THEN
			(* Send_pos	-->	Kommando der fortæller robot cut at nogle nye positioner er sendt *)
			uiSignalOutControl := Send_two_pos;
		END_IF
		IF uiSignalInAck = Send_two_pos THEN
			uiSignalOutControl := 0;
			uiCalibImgCount := uiCalibImgCount + 1;
			NewState := 135;
		END_IF

	135:
		IF uiSignalInAck = 0 THEN
			NewState := 140;
		END_IF

	140: 		(* Grab the stem + Move to image pos *)
		FB_IMAGE_GRAB.Execute := TRUE;
		uiSignalOutControl := FB_IMAGE_GRAB.OutQ;
		IF FB_IMAGE_GRAB.Done THEN
			FB_IMAGE_GRAB.Execute := FALSE;
			NewState := 150;
		END_IF

	150:
		getPickCoords := TRUE;
		IF bPosSentToPcCom AND FB_GET_PICK_COORD.Execute = FALSE THEN
			bPosSentToPcCom := FALSE;
			bGetCoordDone := FALSE;
			NewState := 200;
		END_IF

		(* ------------------------------------------ Move on stem ------------------------------------------ *)

	200:
		IF stDataToVision.CoordXR2G <> 0 AND stDataToVision.CoordYR2G <> 0 AND stDataToVision.CoordZR2G <> 0 THEN
			FB_CAM_TWO_CONTROL.Execute := TRUE;
			IF FB_CAM_TWO_CONTROL.Done THEN
				FB_CAM_TWO_CONTROL.Execute := FALSE;
				(* Check if the stem is found *)
				IF FB_CAM_TWO_CONTROL.StemFound = 1 THEN
					IF FB_CAM_TWO_CONTROL.X > 350 OR FB_CAM_TWO_CONTROL.X < 200 OR FB_CAM_TWO_CONTROL.Y > 350 OR FB_CAM_TWO_CONTROL.Y < 200 THEN
						GviX := 320;
						GviY := 320;
						GviZ := FB_CAM_TWO_CONTROL.Z;
						GviA := 0;
						GviE := 0;
						GviR := 40;
						gResetPcCom := TRUE;
						NewState := 240;
					ELSE
						GviX := FB_CAM_TWO_CONTROL.X;
						GviY := FB_CAM_TWO_CONTROL.Y;
						GviZ := FB_CAM_TWO_CONTROL.Z;
						GviA := 0;
						GviE := 0;
						GviR := 40;
						IF FB_CAM_TWO_CONTROL.JointFound = 1 THEN
							GviPick := FB_CAM_TWO_CONTROL.PickAngle;
							iImageZone := FB_CAM_TWO_CONTROL.Zone;
							gResetPcCom := TRUE;
							NewState := 310;
						ELSE
							gResetPcCom := TRUE;
							NewState := 240;
						END_IF
					END_IF
				ELSE
					gResetPcCom := TRUE;
					NewState := 345;
				END_IF
			END_IF
		END_IF

	240:		(* Send pos to Robots *)
		(* GsendCoord			-->	Starter SendCoordinates sekvensen							-	Sender koordinater til robotterne 		*)
		(* uiSignalOutShared.06	-->	Bekræftelse på at koordinaterne er sendt til udgangene i box 10	-	Acknowledge fra SendCoordinates	*)
		GsendCoord := TRUE;
		IF uiSignalOutShared.06 THEN
			(* Send_pos	-->	Kommando der fortæller robot cut at nogle nye positioner er sendt *)
			uiSignalOutControl := Send_pos;
		END_IF
		IF uiSignalInAck = Send_pos THEN
			uiSignalOutControl := 0;
			uiCalibImgCount := uiCalibImgCount + 1;
			NewState := 245;
		END_IF

	245:
		IF uiSignalInAck = 0 THEN
			NewState := 250;
		END_IF

	250:
		FB_COMOVE_IMAGE.Execute := TRUE;
		uiSignalOutControl := FB_COMOVE_IMAGE.OutQ;
		IF FB_COMOVE_IMAGE.Done THEN
			FB_COMOVE_IMAGE.Execute := FALSE;
			NewState := 260;
		END_IF

	260:
		(* Send Pick coordinate *)
		(* Send Pick pos to PcCom for next image *)
		getPickCoords := TRUE;
		IF bPosSentToPcCom AND FB_GET_PICK_COORD.Execute = FALSE THEN
			bPosSentToPcCom := FALSE;
			NewState := 300;
		END_IF


	(* ------------------------------------------ Find Joint ------------------------------------------ *)

	300:		(* Take a picture *)
		IF stDataToVision.CoordXR2G <> 0 AND stDataToVision.CoordYR2G <> 0 AND stDataToVision.CoordZR2G <> 0 THEN
			FB_CAM_TWO_CONTROL.Execute := TRUE;
			IF FB_CAM_TWO_CONTROL.Done THEN
				IF FB_CAM_TWO_CONTROL.StemFound = 1 THEN
					IF FB_CAM_TWO_CONTROL.X > 350 OR FB_CAM_TWO_CONTROL.X < 200 OR FB_CAM_TWO_CONTROL.Y > 350 OR FB_CAM_TWO_CONTROL.Y < 200 THEN
						GviPick := FB_CAM_TWO_CONTROL.PickAngle;
						IF FB_CAM_TWO_CONTROL.Zone <> 0 THEN
							iImageZone := FB_CAM_TWO_CONTROL.Zone;
						END_IF
						IF FB_CAM_TWO_CONTROL.JointFound = 1 THEN
							GviPick := FB_CAM_TWO_CONTROL.PickAngle;
							FB_CAM_TWO_CONTROL.Execute := FALSE;
							bPosSentToPcCom := FALSE;gResetPcCom := TRUE;
							NewState := 305;
						ELSE
							GviX := 320;
							GviY := 320;
							GviZ := FB_CAM_TWO_CONTROL.Z;
							GviA := 0;
							GviE := 0;
							GviR := 40;
							FB_CAM_TWO_CONTROL.Execute := FALSE;
							gResetPcCom := TRUE;
							NewState := 310;
						END_IF
					ELSE
						GviPick := FB_CAM_TWO_CONTROL.PickAngle;
						IF FB_CAM_TWO_CONTROL.Zone <> 0 THEN
							iImageZone := FB_CAM_TWO_CONTROL.Zone;
						END_IF
						IF FB_CAM_TWO_CONTROL.JointFound = 1 THEN
							GviPick := FB_CAM_TWO_CONTROL.PickAngle;
							bPosSentToPcCom := FALSE;
							FB_CAM_TWO_CONTROL.Execute := FALSE;
							gResetPcCom := TRUE;
							NewState := 305;
						ELSE
							GviX := FB_CAM_TWO_CONTROL.X;
							GviY := FB_CAM_TWO_CONTROL.Y;
							GviZ := FB_CAM_TWO_CONTROL.Z;
							GviA := 0;
							GviE := 0;
							GviR := 40;
							FB_CAM_TWO_CONTROL.Execute := FALSE;
							gResetPcCom := TRUE;
							NewState := 310;
						END_IF
					END_IF
				ELSE
					FB_CAM_TWO_CONTROL.Execute := FALSE;
					gResetPcCom := TRUE;
					NewState := 345;
				END_IF
			END_IF
		END_IF

	305:
		(* Get Cut coord *)
		getCutCoords := TRUE;
		IF bPosSentToPcCom AND FB_GET_CUT_COORD.Execute = FALSE THEN
			bPosSentToPcCom := FALSE;
			NewState := 307;
		END_IF

	307:
		IF uiSignalInAck = 0 THEN
			GviX	:= stDataToVision.CoordXR1G / 10;
			GviY	:= stDataToVision.CoordYR1G / 10;
			GviZ	:= stDataToVision.CoordZR1G / 10;
			gResetPcCom := TRUE;
			NewState := 310;
		END_IF


	310:		(* Send pos *)
		(* GsendCoord			-->	Starter SendCoordinates sekvensen							-	Sender koordinater til robotterne 		*)
		(* uiSignalOutShared.06	-->	Bekræftelse på at koordinaterne er sendt til udgangene i box 10	-	Acknowledge fra SendCoordinates	*)
		GsendCoord := TRUE;
		IF uiSignalOutShared.06 THEN
			(* Send_pos	-->	Kommando der fortæller robot cut at nogle nye positioner er sendt *)
			uiSignalOutControl := Send_pos;
		END_IF
		IF uiSignalInAck = Send_pos THEN
			uiSignalOutControl := 0;
			(*uiCalibImgCount := uiCalibImgCount + 1;*)
			NewState := 315;
		END_IF

	315:
		IF uiSignalInAck = 0 THEN
			IF FB_CAM_TWO_CONTROL.JointFound = 1 THEN
				NewState := 345;
			ELSE
				NewState := 320;
			END_IF
		END_IF

	320:
		FB_COMOVE_IMAGE.Execute := TRUE;
		uiSignalOutControl := FB_COMOVE_IMAGE.OutQ;
		IF FB_COMOVE_IMAGE.Done THEN
			FB_COMOVE_IMAGE.Execute := FALSE;
			NewState := 330;
		END_IF

	330: 		(* Send Pick coordinate *)
		(* Send Pick pos to PcCom for next image *)
		getPickCoords := TRUE;
		IF bPosSentToPcCom AND FB_GET_PICK_COORD.Execute = FALSE THEN
			bPosSentToPcCom := FALSE;
			NewState := 345;
		END_IF

	345:
		IF uiSignalInAck = 0 THEN
			IF stDataFromVision.gJointFound = 1  THEN
				(* Grabbing sequence *)
				gResetPcCom := TRUE;
				NewState := 400;
			ELSIF stDataFromVision.gStemFound = 1 AND stDataFromVision.gJointFound = 0 AND iMoved < 2 THEN
				(* Move further Along stem *)
				NewState := 300;
			ELSIF stDataFromVision.gStemFound = 0 OR iMoved >= 2 THEN
				(* Change configuration *)
				iCnfgChange := iCnfgChange + 1;
				IF uiCalibImgCount >= 50 AND uiCalibImgCount <= 200 THEN
					NewState := 350;
				ELSIF uiCalibImgCount = 250 THEN
					NewState := 450;
				END_IF
				gResetPcCom := TRUE;
				NewState := 350;
			ELSIF stDataFromVision.gJointFound = 255 THEN 	(* If timeout *)
				NewState := 1000;
			END_IF
		END_IF

	(* ------------------------------------------ Change configuration ------------------------------------------ *)
	350:
		IF iCnfgChange <= 5 THEN
			uiCalibImgCount := INT_TO_BYTE(iCnfgChange * 50);
		ELSE
			NewState := 600;
		END_IF
		(* Robot Pick to image pos *)
		FB_PICK_TRUNK_IMAGE.Execute := TRUE;
		uiSignalOutControl := FB_PICK_TRUNK_IMAGE.OutQ;
		IF FB_PICK_TRUNK_IMAGE.Done THEN
			FB_PICK_TRUNK_IMAGE.Execute := FALSE;
			NewState := 360;
		END_IF

	360:		(* Send Pick coordinate *)
		(* Send Pick pos to PcCom for next image *)
		getPickCoords := TRUE;
		IF bPosSentToPcCom THEN
			bPosSentToPcCom := FALSE;
			NewState := 300;
		END_IF


	(* ------------------------------------------ Grab tomatoes ------------------------------------------ *)
	400:		(* Robot Pick grab *)
		FB_PICK_GRAB.Execute := TRUE;
		uiSignalOutControl := FB_PICK_GRAB.OutQ;
		IF FB_PICK_GRAB.Done THEN
			FB_PICK_GRAB.Execute := FALSE;
			NewState := 420;
		END_IF

	420:		(* Cut *)
		FB_RELEASE_CUT.Execute := TRUE;
		IF FB_RELEASE_CUT.Done THEN
			FB_RELEASE_CUT.Execute := FALSE;
			NewState := 425;
		END_IF

	425:		(* Load Cut *)
		FB_LOAD_CUT.Execute := TRUE;
		IF FB_LOAD_CUT.Done THEN
			FB_LOAD_CUT.Execute := FALSE;
			NewState := 430;
		END_IF

	430:		(* Move from pick *)
		FB_PICK_MOVE_FROM_PICK.Execute := TRUE;
		uiSignalOutControl := FB_PICK_MOVE_FROM_PICK.OutQ;
		IF FB_PICK_MOVE_FROM_PICK.Done THEN
			FB_PICK_MOVE_FROM_PICK.Execute := FALSE;
			iMoved := 1;
			NewState := 500;
		END_IF

	(* --------------------------------- DELEAFING ------------------------------------ *)
	500:		(* Image of LEAFS *)
		uiCalibImgCount := INT_TO_BYTE(iMoved * 50);
		FB_PICK_DELEAF_PROGRAM.Execute := TRUE;
		uiSignalOutControl := FB_PICK_DELEAF_PROGRAM.OutQ;
		IF FB_PICK_DELEAF_PROGRAM.Done THEN
			iMoved := iMoved + 1;
			FB_PICK_DELEAF_PROGRAM.Execute := FALSE;
			NewState := 520;
		END_IF

	520:		(* Send Pick coordinate *)
		getPickCoords := TRUE;
		IF bPosSentToPcCom AND FB_GET_PICK_COORD.Execute = FALSE THEN
			bPosSentToPcCom := FALSE;
			NewState := 530;
		END_IF

	530:
		IF stDataToVision.CoordXR2G <> 0 AND stDataToVision.CoordYR2G <> 0 AND stDataToVision.CoordZR2G <> 0 THEN
			FB_CAM_TWO_CONTROL.Execute := TRUE;
			IF FB_CAM_TWO_CONTROL.Done THEN
				IF FB_CAM_TWO_CONTROL.StemFound = 1 THEN
					IF FB_CAM_TWO_CONTROL.X > 500 OR FB_CAM_TWO_CONTROL.X < 200 OR FB_CAM_TWO_CONTROL.Y > 425 OR FB_CAM_TWO_CONTROL.Y < 200 THEN
						FB_CAM_TWO_CONTROL.Execute := FALSE;
						NewState := 1000;
					ELSE
						IF FB_CAM_TWO_CONTROL.JointFound = 1 THEN
							GviX := FB_CAM_TWO_CONTROL.X;
							GviY := FB_CAM_TWO_CONTROL.Y;
							GviZ := FB_CAM_TWO_CONTROL.Z;
							GviA := 0;
							GviE := 0;
							GviR := 40;
							GviPick := FB_CAM_TWO_CONTROL.PickAngle;
							iImageZone := FB_CAM_TWO_CONTROL.Zone;
							gJointFound := FB_CAM_TWO_CONTROL.JointFound;
							FB_CAM_TWO_CONTROL.Execute := FALSE;
							gResetPcCom := TRUE;
							NewState := 540;
						ELSE
							gJointFound := FB_CAM_TWO_CONTROL.JointFound;
							FB_CAM_TWO_CONTROL.Execute := FALSE;
							gResetPcCom := TRUE;
							NewState := 500;
						END_IF
					END_IF
				ELSIF iMoved > 3 THEN
					gJointFound := FB_CAM_TWO_CONTROL.JointFound;
					FB_CAM_TWO_CONTROL.Execute := FALSE;
					gResetPcCom := TRUE;
					NewState := 540;
				ELSE
					FB_CAM_TWO_CONTROL.Execute := FALSE;
					gResetPcCom := TRUE;
					NewState := 500;
				END_IF
			END_IF
		END_IF

	540:		(* Send pos *)
		FB_PLACE.Execute := TRUE;
		IF FB_PLACE.Done THEN
			GviX2 := FB_PLACE.X;
			GviY2 := FB_PLACE.Y;
			GviZ2 := FB_PLACE.Z;
			(* GsendCoord			-->	Starter SendCoordinates sekvensen							-	Sender koordinater til robotterne 		*)
			(* uiSignalOutShared.06	-->	Bekræftelse på at koordinaterne er sendt til udgangene i box 10	-	Acknowledge fra SendCoordinates	*)
			GsendCoord := TRUE;
			IF uiSignalOutShared.06 THEN
				(* Send_pos	-->	Kommando der fortæller robot cut at nogle nye positioner er sendt *)
				uiSignalOutControl := Send_two_pos;
			END_IF
			IF uiSignalInAck = Send_two_pos THEN
				uiSignalOutControl := 0;
				uiCalibImgCount := uiCalibImgCount + 1;
				FB_PLACE.Execute := FALSE;
				NewState := 545;
			END_IF
		END_IF
	545:
		IF uiSignalInAck = 0 THEN
			NewState := 550;
		END_IF

	550:
		FB_PLACE_DELEAF.Execute := TRUE;
		uiSignalOutControl := FB_PLACE_DELEAF.OutQ;
		IF FB_PLACE_DELEAF.Done THEN
			FB_PLACE_DELEAF.Execute := FALSE;
			NewState := 580;
		END_IF

	580:		(* Load Cut *)
		FB_LOAD_CUT.Execute := TRUE;
		IF FB_LOAD_CUT.Done THEN
			FB_LOAD_CUT.Execute := FALSE;
			NewState := 585;
		END_IF

	585:
		IF uiDeleaf < 0 THEN
			uiDeleaf := uiDeleaf + 1;
			NewState := 500;
		ELSE
			uiDeleaf := 0;
			NewState := 600;
		END_IF

	600:		(*Open Cut*)
		FB_OPEN_CUT.Execute := TRUE;
		IF FB_OPEN_CUT.Done THEN
			FB_OPEN_CUT.Execute := FALSE;
			NewState := 610;
		END_IF

	610:		(*Move cut away from stem*)
		FB_CUT_FROM_STEM.Execute := TRUE;
		uiSignalOutControl := FB_CUT_FROM_STEM.OutQ;
		IF FB_CUT_FROM_STEM.Done THEN
			FB_CUT_FROM_STEM.Execute := FALSE;
			NewState := 620;
		END_IF


	620:		(* GbReleaseStem *)
		(* Grab stem and pull in *)
		IF NOT bAck THEN
			(* HMI knap der kalder GribStem *)
			GbReleaseStem := TRUE;
		ELSIF bAck THEN
			NewState := 630;
		END_IF

	630:		(* Move to idle *)
		FB_MOVE_TO_IDLE.Execute := TRUE;
		uiSignalOutControl := FB_MOVE_TO_IDLE.OutQ;
		IF FB_MOVE_TO_IDLE.Done THEN
			FB_MOVE_TO_IDLE.Execute := FALSE;
			uiStatus := 0;
			NewState := 640;
		END_IF

	640:		(* Deload *)

		FB_DELOAD_CUT.Execute := TRUE;
		IF FB_DELOAD_CUT.Done THEN
			FB_DELOAD_CUT.Execute := FALSE;
			NewState := 0;
		END_IF



	1000:	(* Reset *)
		uiSignalOutControl  := 0;		(* Stop sequences on ROBOTS *)
		(* Reset timers *)
		stDataToVision.ResultRead := 1;
		gResetPcCom := TRUE;
		iCnfgChange := 1;
		uiCalibImgCount := 0;
		uiDeleaf := 0;
		NewState := 0;

	2000:
		bStopped := TRUE;

END_CASE

IF State <> 2000 THEN
	bStopped := FALSE;
END_IF

FB_PLACE(Offset := 140,		Box_length := 450, 		Box_width := 400,		Box_height := 125,		Stem_length := 200,	Mode := uiPackingModeNo);

END_PROGRAM

// ---- POUs/FUNCTIONs/PlaceCoordinates.TcPOU
FUNCTION_BLOCK PlaceCoordinates

VAR_INPUT
	Execute: 			BOOL;
	Offset:	 		UINT;
	Box_length:	 	UINT;
	Box_width:		UINT;
	Box_height:		UINT;
	Stem_length:		UINT;
	Reset: 			BOOL;

	Mode: UINT;
END_VAR
VAR_OUTPUT
	X: 				UINT;
	Y: 				UINT;
	Z: 				UINT;
END_VAR

VAR
	(* ARRAYS *)
	PLACE_POS:  ARRAY[1..10000, 1..3] OF UINT :=[ 0,0,0];
	FullArraySize:		UINT;

	(* INTEGERS *)
	State: 			INT := 0;
	NewState: 		INT := 0;
	NewMode:		UINT := 0;

	arraySize: 		UINT;
	arraySize2:		UINT;
	arraySize3: 		UINT;
	counter: 			UINT;
	counter2:			UINT;
	temp:			UINT  := 0;
	i:				UINT;



	(* BOOLS *)
	Done: 			BOOL;
END_VAR

IF State <> NewState THEN
	State := NewState;
END_IF

IF Mode <> NewMode THEN
	NewMode := Mode;
	Reset := TRUE;
END_IF

CASE State OF

	0:		(* INIT	-	Define ARRAY of place positions *)

		IF Mode = 0 THEN
			arraySize := (Box_length - 60) / Offset;
			arraySize2 := (Box_length - 60) / Stem_length;
			FOR i := 1 TO Box_height/20 BY 1 DO
				FOR counter := 1 TO arraySize BY 1 DO
					PLACE_POS[temp + counter, 1] := (Offset * (counter-1)) + 30;
					PLACE_POS[temp + counter, 2] := 30;
					PLACE_POS[temp + counter, 3] := ((i-1) * 30) + 50;
				END_FOR;
				FOR counter := 1 TO arraySize2 BY 1 DO
					PLACE_POS[temp + counter + arraySize, 1] := Offset + 30+ ((counter-1) * Stem_length);
					PLACE_POS[temp + counter + arraySize, 2] := Box_width - 60;
					PLACE_POS[temp + counter + arraySize, 3] := ((i-1) * 30) + 50;
					temp := temp + counter + arraySize;
				END_FOR
			END_FOR
			FullArraySize := (arraySize + arraySize2)*(Box_height/20);
			counter := 1;



		ELSIF Mode = 1 THEN
			ArraySize := (Box_length - 60) / Offset;
			ArraySize2 := 2;
			FOR i := 1 TO Box_height/20 BY 1 DO
				FOR counter := 1 TO ((ArraySize*ArraySize2)-1) BY 2 DO
					PLACE_POS[temp + counter, 1] := (Offset*(counter-1)) + 30;
					PLACE_POS[temp + counter, 2] := 30;
					PLACE_POS[temp + counter, 3] := ((i-1) * 30) + 50;

					PLACE_POS[temp + counter + 1, 1] := (Offset*(counter-1)) + 30;
					PLACE_POS[temp + counter + 1, 2] := Box_width - 30;
					PLACE_POS[temp + counter + 1, 3] := ((i-1) * 30) + 50;
					IF counter >= (ArraySize * ArraySize2)-1 THEN
						temp := temp + counter;
					END_IF
				END_FOR
			END_FOR

			FullArraySize := (Box_height/20) * ((ArraySize*ArraySize2)-1);
			counter := 1;



		ELSIF Mode = 2 THEN
			ArraySize := (Box_length - 60) / Stem_length;
			ArraySize3 := (Box_width - 60) / Offset;
			ArraySize2 := 200 / Offset;
			FOR i := 1 TO Box_height/50 BY 1 DO
				FOR counter := 1 TO ArraySize BY 1 DO
					FOR counter2 := 1 TO ArraySize3 BY 1 DO
						PLACE_POS[temp + counter2, 1] := ((Stem_length/2)*(counter-1)) + 30;
						PLACE_POS[temp + counter2, 2] := (Offset*(counter2-1)) + 30;
						PLACE_POS[temp + counter2, 3] := ((i-1) * 50) + 50;
						IF counter2 = ArraySize3 THEN
							temp := temp + counter2;
						END_IF
					END_FOR
				END_FOR
			END_FOR

			FullArraySize := (Box_height/50) * (ArraySize * ArraySize3);
			counter := 1;

		END_IF

		IF PLACE_POS[FullArraySize, 3] <> 0 THEN
			NewState := 10;
		END_IF


	10:		(* WAIT for Execute *)
		Done := FALSE;
		IF Execute THEN
			NewState := 20;
		END_IF

	20:
		X := PLACE_POS[counter, 1];
		Y := PLACE_POS[counter, 2];
		Z := PLACE_POS[counter, 3];

		NewState := 30;

	30:
		Done := TRUE;

		IF NOT Execute THEN
			IF counter = FullArraySize THEN
				counter := 1;
			ELSE
				counter := counter + 1;
			END_IF
			NewState := 10;
		END_IF

	100:
		FOR i := 1 TO 10000 BY 1 DO
			PLACE_POS[i,1] := 0;
			PLACE_POS[i,2] := 0;
			PLACE_POS[i,3] := 0;
		END_FOR
		IF PLACE_POS[10000, 3] = 0 THEN
			FullArraySize := 0;
			NewState := 0;
		END_IF


END_CASE

IF Reset THEN
	Execute := FALSE;
	temp := 0;
	Counter := 1;
	Reset := FALSE;
	NewState := 100;
END_IF

END_FUNCTION_BLOCK

// ---- POUs/CONTROLs/ControlGrabAuto.TcPOU
PROGRAM ControlGrabAuto
VAR_INPUT
	State: INT := 0;
	NewState: INT := 0;
END_VAR

VAR

	(* INTEGERS *)
	(*uiGripOffset: 		USINT := 220;			(* Offset				-->	Afstand ud til grip, når befinder sig i Home pos	-	Afstand i mm. i Y retning	*)
	uiTrunkPos: 		UINT;				(* Stamme position	-->	Afstand i mm.															*)
	iBunchPosZ: 		UINT;
	iStemAngle:		INT;

	iStemPosX: 		UINT;				(* *)
	iStemPosY: 		UINT;				(* *)
	iStemPosZ: 		UINT;
	iRoll: 			INT;
	iPitch: 			UINT;
	iYaw:			INT;
	iPickAngle: 		INT;*)

	iMoved: 			INT;					(* Hvor mange gange har cut bevæget sig efter iBundPosZ er nået *)
	iCnfgChange:		INT := 0;

	(* REALS *)

	(* Timer *)
	bJointFound: BOOL;
	bStemFound: BOOL;
	flag: BOOL;
	bStopped: BOOL;
	bAngleFlag: BOOL;
	bDeloaded: BOOL;

	uiDeleaf: UINT;
END_VAR

CASE State OF

	0:		(* init	-	Every important variables will be resat before the start of the sequence *)
		IF bStart AND uiprogNo = 5 AND State <> 2000  AND NOT bAlarmState THEN
			uiStatus := 1;

			(* Init variables *)
			uiCalibImgCount	:= 0;
			iMoved := 0;
			iImageZone := 0;
			GviX := 0;
			GviY := 0;
			GviZ := 0;
			GviA := 0;
			GviE := 0;
			GviR := 0;
			GviPick := 0;
			iPickAngle := 0;
			gResetPcCom 	:= TRUE;
			iCnfgChange := 0;
			uiDeleaf := 0;

			(* Before starting - Home *)
			GbHomeGripStem := TRUE;
			IF bHomeDone THEN
				bStart := FALSE;
				bHomeDone := FALSE;
				NewState := 10;
			END_IF
		END_IF

	10:		(* Set velocity *)
		uiSignalOutSpeedControl := UINT_TO_BYTE(uiSpeedSetting);
		FB_SET_VELOCITY.Execute := TRUE;
		uiSignalOutControl := FB_SET_VELOCITY.OutQ;
		IF FB_SET_VELOCITY.Done THEN
			FB_SET_VELOCITY.Execute := FALSE;
			NewState := 20;
		END_IF

	20:		(* Idle *)
		FB_MOVE_TO_IDLE.Execute := TRUE;
		uiSignalOutControl := FB_MOVE_TO_IDLE.OutQ;
		IF FB_MOVE_TO_IDLE.Done THEN
			FB_MOVE_TO_IDLE.Execute := FALSE;
			NewState := 30;
		END_IF

	30:		(*  Load cutter *)
		FB_LOAD_CUT.Execute := TRUE;
		IF FB_LOAD_CUT.Done THEN
			FB_LOAD_CUT.Execute := FALSE;
			NewState := 40;
		END_IF

	40: 		(* Cam 1 Take image	-	parameters recieved from Vision = height of lowest ripe tomato and Y coord for lowest point of the stem *)

		FB_CAM_ONE_CONTROL.Execute := TRUE;
		IF FB_CAM_ONE_CONTROL.Done THEN
			FB_CAM_ONE_CONTROL.Execute := FALSE;

			uiDistToGrab	:= FB_CAM_ONE_CONTROL.TrunkDist;
			iBunchPosZ 	:= FB_CAM_ONE_CONTROL.BunchHeight;
			iStemAngle	:= FB_CAM_ONE_CONTROL.StemHeading;
			iImageZone	:= FB_CAM_ONE_CONTROL.Zone;
			NewState := 50;
		END_IF

	50:		(* Joris gripper retreives stem *)
		(* Grab stem and pull in *)
		IF NOT bAck THEN
			(* HMI knap der kalder GribStem *)
			GbGripStem := TRUE;
		ELSIF bAck THEN
			gResetPcCom := TRUE;
			NewState := 55;
		END_IF

	55:
		IF uiToolState = 0 THEN
			NewState := 100;
		END_IF

	(* ---------------------------- Grab the stem ---------------------------- *)

	100:		(* Robot Pick move to Image Pos *)
		FB_PICK_TRUNK_IMAGE.Execute := TRUE;
		uiSignalOutControl := FB_PICK_TRUNK_IMAGE.OutQ;
		IF FB_PICK_TRUNK_IMAGE.Done THEN
			FB_PICK_TRUNK_IMAGE.Execute := FALSE;
			gResetPcCom := TRUE;
			NewState := 110;
		END_IF

	110:		(* Send Robot Pick Position *)
		getPickCoords := TRUE;
		IF bPosSentToPcCom AND FB_GET_PICK_COORD.Execute = FALSE THEN
			bPosSentToPcCom := FALSE;
			bGetCoordDone := FALSE;
			NewState := 120;
		END_IF

	120:		(* Cam 2 take image *)
		(* Take bottom Image *)
		IF stDataToVision.CoordXR2G <> 0 AND stDataToVision.CoordYR2G <> 0 AND stDataToVision.CoordZR2G <> 0 THEN
			FB_CAM_TWO_CONTROL.Execute := TRUE;
			IF FB_CAM_TWO_CONTROL.Done THEN
				FB_CAM_TWO_CONTROL.Execute := FALSE;
				IF FB_CAM_TWO_CONTROL.X > 420 OR FB_CAM_TWO_CONTROL.X < 125 OR FB_CAM_TWO_CONTROL.Y > 400 OR FB_CAM_TWO_CONTROL.Y < 125 THEN
					NewState := 1000;
				ELSE
					GviX := FB_CAM_TWO_CONTROL.X;
					GviY := FB_CAM_TWO_CONTROL.Y;
					GviZ := FB_CAM_TWO_CONTROL.Z;
					GviA := FB_CAM_TWO_CONTROL.RotZ0;
					GviE := FB_CAM_TWO_CONTROL.RotY;
					GviR := FB_CAM_TWO_CONTROL.RotZ1;
					gResetPcCom := TRUE;
					NewState := 130;
				END_IF
			END_IF
		END_IF

	130:		(* Send Pos to Robot *)

		(* GsendCoord			-->	Starter SendCoordinates sekvensen							-	Sender koordinater til robotterne 		*)
		(* uiSignalOutShared.06	-->	Bekræftelse på at koordinaterne er sendt til udgangene i box 10	-	Acknowledge fra SendCoordinates	*)
		GsendCoord := TRUE;
		IF uiSignalOutShared.06 THEN
			(* Send_pos	-->	Kommando der fortæller robot cut at nogle nye positioner er sendt *)
			uiSignalOutControl := Send_pos;
		END_IF
		IF uiSignalInAck = Send_pos THEN
			uiSignalOutControl := 0;
			uiCalibImgCount := uiCalibImgCount + 1;
			NewState := 135;
		END_IF

	135:
		IF uiSignalInAck = 0 THEN
			NewState := 140;
		END_IF

	140:		(* Move Pick to next image pos *)
		FB_PICK_TRUNK_IMAGE.Execute := TRUE;
		uiSignalOutControl := FB_PICK_TRUNK_IMAGE.OutQ;
		IF FB_PICK_TRUNK_IMAGE.Done THEN
			FB_PICK_TRUNK_IMAGE.Execute := FALSE;
			NewState := 150;
		END_IF

	150:		(* Send Pick pos to PcCom for next image *)
		getPickCoords := TRUE;
		IF bPosSentToPcCom AND FB_GET_PICK_COORD.Execute = FALSE THEN
			bPosSentToPcCom := FALSE;
			bGetCoordDone := FALSE;
			NewState := 160;
		END_IF

	160:		(* Move Cut to Stem *)
		FB_CUT_TO_STEM.Execute := TRUE;
		uiSignalOutControl := FB_CUT_TO_STEM.OutQ;
		IF FB_CUT_TO_STEM.Done THEN
			FB_CUT_TO_STEM.Execute := FALSE;
			IF FB_CAM_TWO_CONTROL.Z >= iBunchPosZ THEN
				NewState := 300;
			ELSE
				NewState := 200;
			END_IF
		END_IF

		(* ------------------------------------------ Move on stem ------------------------------------------ *)

	200:		(* Cam 2: Take new Image *)
		IF stDataToVision.CoordXR2G <> 0 AND stDataToVision.CoordYR2G <> 0 AND stDataToVision.CoordZR2G <> 0 THEN
			FB_CAM_TWO_CONTROL.Execute := TRUE;
			IF FB_CAM_TWO_CONTROL.Done THEN
				FB_CAM_TWO_CONTROL.Execute := FALSE;
				IF FB_CAM_TWO_CONTROL.StemFound = 1 THEN
					IF FB_CAM_TWO_CONTROL.X > 500 OR FB_CAM_TWO_CONTROL.X < 125 OR FB_CAM_TWO_CONTROL.Y > 425 OR FB_CAM_TWO_CONTROL.Y < 125 THEN
						NewState := 1000;
					ELSE
						GviX := FB_CAM_TWO_CONTROL.X;
						GviY := FB_CAM_TWO_CONTROL.Y;
						GviZ := FB_CAM_TWO_CONTROL.Z;
						GviA := 0;
						GviE := 0;
						GviR := 40;
						IF FB_CAM_TWO_CONTROL.JointFound = 1 THEN
							GviPick := FB_CAM_TWO_CONTROL.PickAngle;
							iImageZone := FB_CAM_TWO_CONTROL.Zone;
							gResetPcCom := TRUE;
							NewState := 310;
						ELSE
							gResetPcCom := TRUE;
							NewState := 210;
						END_IF
					END_IF
				ELSE
					gResetPcCom := TRUE;
					NewState := 345;
				END_IF
			END_IF
		END_IF

	210:		(* Send pos to Robots *)
		(* GsendCoord			-->	Starter SendCoordinates sekvensen							-	Sender koordinater til robotterne 		*)
		(* uiSignalOutShared.06	-->	Bekræftelse på at koordinaterne er sendt til udgangene i box 10	-	Acknowledge fra SendCoordinates	*)
		GsendCoord := TRUE;
		IF uiSignalOutShared.06 THEN
			(* Send_pos	-->	Kommando der fortæller robot cut at nogle nye positioner er sendt *)
			uiSignalOutControl := Send_pos;
		END_IF
		IF uiSignalInAck = Send_pos THEN
			uiSignalOutControl := 0;
			uiCalibImgCount := uiCalibImgCount + 1;
			NewState := 215;
		END_IF

	215:
		IF uiSignalInAck = 0 THEN
			NewState := 220;
		END_IF

	220:		(* Robot Pick to image pos *)
		FB_PICK_TRUNK_IMAGE.Execute := TRUE;
		uiSignalOutControl := FB_PICK_TRUNK_IMAGE.OutQ;
		IF FB_PICK_TRUNK_IMAGE.Done THEN
			FB_PICK_TRUNK_IMAGE.Execute := FALSE;
			NewState := 230;
		END_IF

	230: 		(* Send Pick coordinate *)
		(* Send Pick pos to PcCom for next image *)
		getPickCoords := TRUE;
		IF bPosSentToPcCom AND FB_GET_PICK_COORD.Execute = FALSE THEN
			bPosSentToPcCom := FALSE;
			NewState := 240;
		END_IF

	240:		(* Move cut on stem *)
		FB_CUT_ON_STEM.Execute := TRUE;
		uiSignalOutControl := FB_CUT_ON_STEM.OutQ;
		(* MOVE_TO_STEM bliver sendt tilbage som bekræftelse *)
		IF FB_CUT_ON_STEM.Done THEN
			FB_CUT_ON_STEM.Execute := FALSE;
			IF iStemPosZ >= iBunchPosZ THEN
				iMoved := 0;
				NewState := 300;
			ELSE
				NewState := 200;
			END_IF
		END_IF

	(* ------------------------------------------ Find Joint ------------------------------------------ *)

	300:		(* Take a picture *)
		IF stDataToVision.CoordXR2G <> 0 AND stDataToVision.CoordYR2G <> 0 AND stDataToVision.CoordZR2G <> 0 THEN
			FB_CAM_TWO_CONTROL.Execute := TRUE;
			IF FB_CAM_TWO_CONTROL.Done THEN
				FB_CAM_TWO_CONTROL.Execute := FALSE;
				IF FB_CAM_TWO_CONTROL.StemFound = 1 THEN
					IF FB_CAM_TWO_CONTROL.X > 500 OR FB_CAM_TWO_CONTROL.X < 125 OR FB_CAM_TWO_CONTROL.Y > 425 OR FB_CAM_TWO_CONTROL.Y < 125 THEN
						NewState := 1000;
					ELSE
						GviPick := FB_CAM_TWO_CONTROL.PickAngle;
						IF FB_CAM_TWO_CONTROL.Zone <> 0 THEN
							iImageZone := FB_CAM_TWO_CONTROL.Zone;
						END_IF
						IF FB_CAM_TWO_CONTROL.JointFound = 1 THEN
							GviPick := FB_CAM_TWO_CONTROL.PickAngle;
						ELSE
							GviX := FB_CAM_TWO_CONTROL.X;
							GviY := FB_CAM_TWO_CONTROL.Y;
							GviZ := FB_CAM_TWO_CONTROL.Z;
							GviA := 0;
							GviE := 0;
							GviR := 40;
						END_IF
						gResetPcCom := TRUE;
						NewState := 310;
					END_IF
				ELSE
					gResetPcCom := TRUE;
					NewState := 345;
				END_IF
			END_IF
		END_IF

	310:		(* Send pos *)
		(* GsendCoord			-->	Starter SendCoordinates sekvensen							-	Sender koordinater til robotterne 		*)
		(* uiSignalOutShared.06	-->	Bekræftelse på at koordinaterne er sendt til udgangene i box 10	-	Acknowledge fra SendCoordinates	*)
		GsendCoord := TRUE;
		IF uiSignalOutShared.06 THEN
			(* Send_pos	-->	Kommando der fortæller robot cut at nogle nye positioner er sendt *)
			uiSignalOutControl := Send_pos;
		END_IF
		IF uiSignalInAck = Send_pos THEN
			uiSignalOutControl := 0;
			uiCalibImgCount := uiCalibImgCount + 1;
			bAngleFlag := FALSE;
			NewState := 315;
		END_IF

	315:
		IF uiSignalInAck = 0 THEN
			IF FB_CAM_TWO_CONTROL.JointFound = 1 THEN
				NewState := 345;
			ELSE
				NewState := 320;
			END_IF
		END_IF

	320:		(* Pick image pos *)
		(* Robot Pick to image pos *)
		FB_PICK_TRUNK_IMAGE.Execute := TRUE;
		uiSignalOutControl := FB_PICK_TRUNK_IMAGE.OutQ;
		IF FB_PICK_TRUNK_IMAGE.Done THEN
			FB_PICK_TRUNK_IMAGE.Execute := FALSE;
			NewState := 330;
		END_IF

	330: 		(* Send Pick coordinate *)
		(* Send Pick pos to PcCom for next image *)
		getPickCoords := TRUE;
		IF bPosSentToPcCom AND FB_GET_PICK_COORD.Execute = FALSE THEN
			bPosSentToPcCom := FALSE;
			NewState := 340;
		END_IF

	340:		(* Move on Stem *)
		FB_CUT_ON_STEM.Execute := TRUE;
		uiSignalOutControl := FB_CUT_ON_STEM.OutQ;
		(* MOVE_TO_STEM bliver sendt tilbage som bekræftelse *)
		IF FB_CUT_ON_STEM.Done THEN
			FB_CUT_ON_STEM.Execute := FALSE;
			iCnfgChange := 0;
			iMoved := iMoved +1;
			NewState := 345;
		END_IF

	345:
		IF uiSignalInAck = 0 THEN
			IF stDataFromVision.gJointFound = 1  THEN
				(* Grabbing sequence *)
				gResetPcCom := TRUE;
				NewState := 400;
			ELSIF stDataFromVision.gStemFound = 1 AND stDataFromVision.gJointFound = 0 AND iMoved < 2 THEN
				(* Move further Along stem *)
				NewState := 300;
			ELSIF stDataFromVision.gStemFound = 0 OR iMoved >= 2 THEN
				(* Change configuration *)
				iCnfgChange := iCnfgChange + 1;
				IF uiCalibImgCount >= 50 AND uiCalibImgCount <= 200 THEN
					NewState := 350;
				ELSIF uiCalibImgCount = 250 THEN
					NewState := 450;
				END_IF
				gResetPcCom := TRUE;
				NewState := 350;
			ELSIF stDataFromVision.gJointFound = 255 THEN 	(* If timeout *)
				NewState := 1000;
			END_IF
		END_IF

	(* ------------------------------------------ Change configuration ------------------------------------------ *)
	350:
		IF iCnfgChange <= 5 THEN
			uiCalibImgCount := INT_TO_BYTE(iCnfgChange * 50);
		ELSE
			NewState := 600;
		END_IF
		(* Robot Pick to image pos *)
		FB_PICK_TRUNK_IMAGE.Execute := TRUE;
		uiSignalOutControl := FB_PICK_TRUNK_IMAGE.OutQ;
		IF FB_PICK_TRUNK_IMAGE.Done THEN
			FB_PICK_TRUNK_IMAGE.Execute := FALSE;
			NewState := 360;
		END_IF

	360:		(* Send Pick coordinate *)
		(* Send Pick pos to PcCom for next image *)
		getPickCoords := TRUE;
		IF bPosSentToPcCom THEN
			bPosSentToPcCom := FALSE;
			NewState := 300;
		END_IF


	(* ------------------------------------------ Grab tomatoes ------------------------------------------ *)
	400:		(* Robot Pick grab *)
		FB_PICK_GRAB.Execute := TRUE;
		uiSignalOutControl := FB_PICK_GRAB.OutQ;
		IF FB_PICK_GRAB.Done THEN
			FB_PICK_GRAB.Execute := FALSE;
			NewState := 420;
		END_IF

	420:		(* Cut *)
		FB_RELEASE_CUT.Execute := TRUE;
		IF FB_RELEASE_CUT.Done THEN
			FB_RELEASE_CUT.Execute := FALSE;
			NewState := 425;
		END_IF

	425:		(* Load Cut *)
		FB_LOAD_CUT.Execute := TRUE;
		IF FB_LOAD_CUT.Done THEN
			FB_LOAD_CUT.Execute := FALSE;
			NewState := 430;
		END_IF

	430:		(* Move from pick *)
		FB_PICK_MOVE_FROM_PICK.Execute := TRUE;
		uiSignalOutControl := FB_PICK_MOVE_FROM_PICK.OutQ;
		IF FB_PICK_MOVE_FROM_PICK.Done THEN
			FB_PICK_MOVE_FROM_PICK.Execute := FALSE;
			iMoved := 1;
			NewState := 500;
		END_IF

	(* --------------------------------- DELEAFING ------------------------------------ *)
	500:		(* Image of LEAFS *)
		uiCalibImgCount := INT_TO_BYTE(iMoved * 50);
		FB_PICK_DELEAF_PROGRAM.Execute := TRUE;
		uiSignalOutControl := FB_PICK_DELEAF_PROGRAM.OutQ;
		IF FB_PICK_DELEAF_PROGRAM.Done THEN
			iMoved := iMoved + 1;
			FB_PICK_DELEAF_PROGRAM.Execute := FALSE;
			NewState := 520;
		END_IF

	520:		(* Send Pick coordinate *)
		getPickCoords := TRUE;
		IF bPosSentToPcCom AND FB_GET_PICK_COORD.Execute = FALSE THEN
			bPosSentToPcCom := FALSE;
			NewState := 530;
		END_IF

	530:
		IF stDataToVision.CoordXR2G <> 0 AND stDataToVision.CoordYR2G <> 0 AND stDataToVision.CoordZR2G <> 0 THEN
			FB_CAM_TWO_CONTROL.Execute := TRUE;
			IF FB_CAM_TWO_CONTROL.Done THEN
				FB_CAM_TWO_CONTROL.Execute := FALSE;

				IF FB_CAM_TWO_CONTROL.StemFound = 1 THEN
					IF FB_CAM_TWO_CONTROL.X > 500 OR FB_CAM_TWO_CONTROL.X < 125 OR FB_CAM_TWO_CONTROL.Y > 425 OR FB_CAM_TWO_CONTROL.Y < 125 THEN
						NewState := 1000;
					ELSE
						IF FB_CAM_TWO_CONTROL.JointFound = 1 THEN
							GviX := FB_CAM_TWO_CONTROL.X;
							GviY := FB_CAM_TWO_CONTROL.Y;
							GviZ := FB_CAM_TWO_CONTROL.Z;
							GviA := 0;
							GviE := 0;
							GviR := 40;
							GviPick := FB_CAM_TWO_CONTROL.PickAngle;
							iImageZone := FB_CAM_TWO_CONTROL.Zone;
							gResetPcCom := TRUE;
							NewState := 540;
						ELSE
							gResetPcCom := TRUE;
							NewState := 500;
						END_IF
					END_IF
				ELSIF iMoved > 3 THEN
					gResetPcCom := TRUE;
					NewState := 540;

				ELSE
					gResetPcCom := TRUE;
					NewState := 500;
				END_IF
			END_IF
		END_IF

	540:		(* Cut move on stem *)
		FB_PICK_PLACE.Execute := TRUE;
		uiSignalOutControl := FB_PICK_PLACE.OutQ;
		IF FB_PICK_PLACE.Done THEN
			FB_PICK_PLACE.Execute := FALSE;
			stDataToVision.ResultRead := 0;
			gResetPcCom := TRUE;
			IF FB_CAM_TWO_CONTROL.JointFound = 0 THEN
				NewState := 600;
			ELSE
				NewState := 550;
			END_IF
		END_IF

	550:		(* Send pos *)

		(* GsendCoord			-->	Starter SendCoordinates sekvensen							-	Sender koordinater til robotterne 		*)
		(* uiSignalOutShared.06	-->	Bekræftelse på at koordinaterne er sendt til udgangene i box 10	-	Acknowledge fra SendCoordinates	*)
		GsendCoord := TRUE;
		IF uiSignalOutShared.06 THEN
			(* Send_pos	-->	Kommando der fortæller robot cut at nogle nye positioner er sendt *)
			uiSignalOutControl := Send_pos;
		END_IF
		IF uiSignalInAck = Send_pos THEN
			uiSignalOutControl := 0;
			uiCalibImgCount := uiCalibImgCount + 1;
			NewState := 560;
		END_IF
	560:
		FB_CUT_ON_STEM.Execute := TRUE;
		uiSignalOutControl := FB_CUT_ON_STEM.OutQ;
		IF FB_CUT_ON_STEM.Done THEN
			FB_CUT_ON_STEM.Execute := FALSE;
			NewState := 570;
		END_IF

	570:		(* CUT *)
		FB_RELEASE_CUT.Execute := TRUE;
		IF FB_RELEASE_CUT.Done THEN
			FB_RELEASE_CUT.Execute := FALSE;
			NewState := 580;
		END_IF

	580:		(* Load Cut *)
		FB_LOAD_CUT.Execute := TRUE;
		IF FB_LOAD_CUT.Done THEN
			FB_LOAD_CUT.Execute := FALSE;
			NewState := 585;
		END_IF

	585:
		IF uiDeleaf < 0 THEN
			uiDeleaf := uiDeleaf + 1;
			NewState := 500;
		ELSE
			uiDeleaf := 0;
			NewState := 600;
		END_IF

	600:		(*Open Cut*)
		FB_OPEN_CUT.Execute := TRUE;
		IF FB_OPEN_CUT.Done THEN
			FB_OPEN_CUT.Execute := FALSE;
			NewState := 610;
		END_IF

	610:		(*Move cut away from stem*)
		FB_CUT_FROM_STEM.Execute := TRUE;
		uiSignalOutControl := FB_CUT_FROM_STEM.OutQ;
		IF FB_CUT_FROM_STEM.Done THEN
			FB_CUT_FROM_STEM.Execute := FALSE;
			NewState := 620;
		END_IF


	620:		(* GbReleaseStem *)
		(* Grab stem and pull in *)
		IF NOT bAck THEN
			(* HMI knap der kalder GribStem *)
			GbReleaseStem := TRUE;
		ELSIF bAck THEN
			NewState := 630;
		END_IF

	630:		(* Move to idle *)
		FB_MOVE_TO_IDLE.Execute := TRUE;
		uiSignalOutControl := FB_MOVE_TO_IDLE.OutQ;
		IF FB_MOVE_TO_IDLE.Done THEN
			FB_MOVE_TO_IDLE.Execute := FALSE;
			uiStatus := 0;
			NewState := 640;
		END_IF

	640:		(* Deload *)

		FB_DELOAD_CUT.Execute := TRUE;
		IF FB_DELOAD_CUT.Done THEN
			FB_DELOAD_CUT.Execute := FALSE;
			NewState := 0;
		END_IF



	1000:	(* Reset *)
		uiSignalOutControl  := 0;		(* Stop sequences on ROBOTS *)
		FB_CAM_ONE_CONTROL.	Execute := FALSE;
		FB_CAM_TWO_CONTROL.	Execute := FALSE;
		(* Reset timers *)
		stDataToVision.ResultRead := 1;
		gResetPcCom := TRUE;
		bDeloaded := FALSE;
		iCnfgChange := 1;
		uiCalibImgCount := 0;
		uiDeleaf := 0;
		NewState := 0;

	2000:
		bStopped := TRUE;

END_CASE

IF State <> 2000 THEN
	bStopped := FALSE;
END_IF

END_PROGRAM

// ---- POUs/CONTROLs/ControlMoveToCalibPos.TcPOU
PROGRAM ControlMoveToCalibPos
VAR_INPUT
	State: INT := 0;
	NewState: INT := 0;
END_VAR

VAR

	(* Timer *)
	Wait:TON;
	WaitCut:TON;

	test: BOOL;

	counter: INT := 0;
	bWait: BOOL;
	bWaitCut: BOOL;
	testX: INT;
	testY: INT;
	testCount: INT := 0;
	Wait2: TON;
	Wait3: TON;
	bWait2: BOOL;
	next: BOOL;
	bWait3: BOOL;
	bStopped: BOOL;
	iBottomPosY: INT;
	iBottomPosX: INT;
	iBottomPosZ: INT;
	iTopPosX: INT;
	iTopPosY: INT;
	iTopPosZ: INT;
	bResetSat: BOOL;
	rDotZY: REAL;
	rDotZX: REAL;
	rDotYX: REAL;
	rMagnitudeZY: REAL;
	rMagnitudeZX: REAL;
	rMagnitudeYX: REAL;
	iAngleZY: REAL;
	iAngleZX: REAL;
	iAngleYX: REAL;

	iUnity:	ARRAY[0..2] OF INT :=[ 0, 0, 1];
	iOriVec:	ARRAY[0..2] OF INT;
	bConverted: BOOL;
	iRoll: INT;
	iPitch: INT;
	iYaw: INT;
END_VAR

CASE State OF

	0:		(* Move robot pick to pos from sequence 14 *)
		uiStatus := 0;
		IF bStart AND uiprogNo = 3 AND State <> 2000  AND NOT bAlarmState THEN
			uiStatus := 1;
			Cam := FALSE;
			(* Encoder	-->	Så grip kan køre til den korrekte position *)
			(* Before starting - Home *)
			GbHomeGripStem := TRUE;
			IF bHomeDone THEN
				bHomeDone := FALSE;
				NewState := 5;
			END_IF
		END_IF

	5:		(* Velocity *)
   		uiSignalOutSpeedControl := UINT_TO_BYTE(uiSpeedSetting);
		uiSignalOutControl := Set_Velocity;
		IF uiSignalInAck = Set_Velocity THEN
			uiSignalOutControl := 0;
			NewState := 10;
		END_IF

	10:		(* Move to Idle positions *)
		IF uiSignalInAck = 0 THEN
			NewState := 15;
		END_IF

	15:		(* Get pick coord *)

		(* Before the picture is taken, call get pick coord *)
		getPickCoords := TRUE;
		IF uiSignalInAck = getCurrentPickCoords THEN
			uiSignalOutControl := 0;
			NewState := 17;
		END_IF

	17:
		uiSignalOutControl := 0;
		IF uiSignalInAck = 0 THEN
			IF bPosSentToPcCom THEN
				stDataToVision.ResultRead := 0;
				bPosSentToPcCom := FALSE;
				bGetCoordDone := FALSE;
				NewState := 30;
			END_IF
		END_IF

	20:		(* GET position from PC for robot pick *)

		IF stDataToVision.CoordXR2G <> 0 AND stDataToVision.CoordYR2G <> 0 AND stDataToVision.CoordZR2G <> 0 THEN
			IF Cam THEN
				bTestCamPointCam1 := TRUE;										(* Sends CmdByte 14 to PC *)
			ELSE
				bTestCamPointCam2 := TRUE;
			END_IF
			IF stDataFromVision.CmdInProcess = stDataToVision.CmdByte AND stDataToVision.CmdByte <> 0 THEN					(* When the PC  has sent the position, prepare to send the position to robot pick *)
				iBottomPosX 	:= stDataFromVision.ResultPar1;
				iBottomPosY 	:= stDataFromVision.ResultPar2;
				iBottomPosZ 	:= stDataFromVision.ResultPar3;
				
				bTestCamPointCam1 := FALSE;
				bTestCamPointCam2 := FALSE;
				NewState := 25;
			END_IF
		END_IF

	25:		(*Reset PcCom Values *)
		(* Når ResultReady også sættes lav *)
		stDataToVision.ResultRead := 0;
		NewState := 30;

	30:		(* Take Top Image *)
		IF stDataToVision.CoordXR2G <> 0 AND stDataToVision.CoordYR2G <> 0 AND stDataToVision.CoordZR2G <> 0 THEN
			IF Cam THEN
				bTestCamPointCam1 := TRUE;										(* Sends CmdByte 14 to PC *)
			ELSE
				bTestCamPointCam2 := TRUE;
			END_IF									(* Send CmdByte 14 to PC *)
			IF stDataFromVision.CmdInProcess = stDataToVision.CmdByte AND stDataToVision.CmdByte <> 0 THEN					(* When the PC  has sent the position, prepare to send the position to robot pick *)
				iTopPosX 	:= stDataFromVision.ResultPar1;
				iTopPosY 	:= stDataFromVision.ResultPar2;
				iTopPosZ 	:= stDataFromVision.ResultPar3;
				iRoll	 		:= stDataFromVision.ResultPar4;
				iPitch		:= stDataFromVision.ResultPar5;
				iYaw		:= stDataFromVision.ResultPar6;

				bTestCamPointCam1 := FALSE;
				bTestCamPointCam2 := FALSE;
				NewState := 35;
			END_IF
		END_IF

	35:		(*Reset PcCom Values *)
		(* Når ResultReady også sættes lav *)
		bWaitCut := TRUE;
		IF WaitCut.Q THEN
			IF NOT bResetSat THEN
				bResetSat := TRUE;
				gResetPcCom := TRUE;
			END_IF
			IF NOT gResetPcCom  THEN
				bWaitCut := FALSE;
				bResetSat := FALSE;
				NewState := 50;
			END_IF
		END_IF

	40:		(* Calculate Angles *)
		(* Angle between two vectors are: cos(theta) = [U*V / (||U|| * ||V||)]	=>	theta =cos^-1[U*V / (||U|| * ||V||)] 		*)
		(* Assume both vectors start in 0	-->	Magnitude = arrVector[0..2]										*)

		iOriVec[0] := iBottomPosX - iTopPosX;
		iOriVec[1] := iBottomPosY - iTopPosY;
		iOriVec[2] := iBottomPosZ - iTopPosZ;

		rDotZY := (iOriVec[1] * iUnity[1]) + (iOriVec[2] * iUnity[2]);
		rDotZX := (iOriVec[0] * iUnity[0]) + (iOriVec[2] * iUnity[2]);
		rDotYX := (iOriVec[0] * iUnity[0]) + (iOriVec[1] * iUnity[1]);

		rMagnitudeZY := SQRT((iOriVec[2] * iOriVec[2]) + (iOriVec[1] * iOriVec[1])) * SQRT((iUnity[2] * iUnity[2]) + (iUnity[1] * iUnity[1]));
		rMagnitudeZX := SQRT((iOriVec[2] * iOriVec[2]) + (iOriVec[0] * iOriVec[0])) * SQRT((iUnity[2] * iUnity[2]) + (iUnity[0] * iUnity[0]));
		rMagnitudeYX := SQRT((iOriVec[1] * iOriVec[1]) + (iOriVec[0] * iOriVec[0])) * SQRT((iUnity[1] * iUnity[1]) + (iUnity[0] * iUnity[0]));

		(* Angle = ACOS(DOT_PRODUCT / MAGNITUDE) *)
		(* Angle between Z and Y *)
		iAngleZY := ACOS( (rDotZY) / rMagnitudeZY);
		(* Angle between Z and X *)
		iAngleZX := ACOS( (rDotZX) / rMagnitudeZX);
		(* Angle between Y and X *)
		iAngleYX := ACOS( (rDotYX) / rMagnitudeYX);

		NewState := 45;

	45:
		(* Convert from radians to degrees *)
		IF NOT bConverted THEN
			iAngleZY := (iAngleZY * (180/3.1415)) - 180;
			iAngleZX := (iAngleZX * (180/3.1415))  - 180;
			iAngleYX := (iAngleYX * (180/3.1415)) - 180;
			bConverted := TRUE;
		END_IF
		IF bConverted THEN
			NewState := 50;
		END_IF

	50:		(* Send Pos to Robot *)
		bConverted := FALSE;
		GviX := iTopPosX;	(*(iBottomPosX + iTopPosX) / 2;*)
		GviY := iTopPosY;	(*(iBottomPosY + iTopPosY) / 2;*)
		GviZ := iTopPosZ;	(*(iBottomPosZ + iTopPosZ) / 2;*)
		GviA := REAL_TO_INT(iRoll);
		GviE := REAL_TO_INT(iPitch);
		GviR :=REAL_TO_INT(stDataFromVision.ResultPar6);

		(* GsendCoord			-->	Starter SendCoordinates sekvensen							-	Sender koordinater til robotterne 		*)
		(* uiSignalOutShared.06	-->	Bekræftelse på at koordinaterne er sendt til udgangene i box 10	-	Acknowledge fra SendCoordinates	*)
		GsendCoord := TRUE;
		IF uiSignalOutShared.06 THEN
			(* Send_pos	-->	Kommando der fortæller robot cut at nogle nye positioner er sendt *)
			uiSignalOutControl := Send_pos;
		END_IF
		IF uiSignalInAck = Send_pos THEN
			uiSignalOutControl := 0;
			NewState := 55;
		END_IF

	55:
		IF uiSignalInAck = 0 THEN
			NewState := 60;
		END_IF

	60:		(* Move Pick to the position *)
		IF Cam THEN
			uiSignalOutControl := Pick_Move_To_Pos;
			IF uiSignalInAck = Pick_Move_To_Pos THEN
				uiSignalOutControl := 0;
				NewState := 65;
			END_IF
		ELSE
			uiSignalOutControl := MOVE_CUT_TO_POS;
			IF uiSignalInAck = MOVE_CUT_TO_POS THEN
				uiSignalOutControl := 0;
				NewState := 65;
			END_IF
		END_IF

	65:
		IF next THEN
			next := FALSE;
			uiSignalOutControl := 0;
			NewState := 70;
		END_IF

	70:		(* Move to idle *)
		uiSignalOutControl := Move_to_idle;
		IF uiSignalInAck = Move_to_idle THEN
			uiSignalOutControl := 0;
			uiStatus := 0;
			Cam := FALSE;
			NewState := 0;
		END_IF

	1000:		(* RESET *)
		test 					:= FALSE;
		getPickCoords 		:= FALSE;
		bWait 				:= FALSE;
		bWait2 				:= FALSE;
		bWait3 				:= FALSE;
		uiSignalOutControl 	:= 0;
		bTestCamPointCam1 	:= FALSE;
		bTestCamPointCam2 	:= FALSE;
		next 					:= FALSE;
		uiSignalOutShared.06 	:= FALSE;

		NewState := 0;

	2000:
		bStopped := TRUE;

END_CASE

IF State <> 2000 THEN
	bStopped := FALSE;
END_IF

(*  ______________________________________________________________________ *)

Wait		(IN:=  bWait		, PT:=t#200ms, Q=>, ET=>); 			(*Timer*)
WaitCut	(IN:=  bWaitCut		, PT:=t#1000ms, Q=>, ET=>); 	(*Timer*)
Wait2	(IN:=  bWait2		, PT:=t#2000ms, Q=>, ET=>); 		(*Timer*)
Wait3	(IN:=  bWait3		, PT:=t#500ms, Q=>, ET=>); 		(*Timer*)

END_PROGRAM

// ---- POUs/SendCoordinates.TcPOU
PROGRAM SendCoordinates
VAR_INPUT
	State: INT :=0;
END_VAR

VAR

	viX: INT;
	viY: INT;
	viZ: INT;
	viA: INT;
	viE: INT;
	viR: INT;

	NewState: INT := 0;
END_VAR

(* SendCoordinates	-->	Sender Koordinater fra PLC til Robot *)

CASE State OF

	0:
		IF GsendCoord THEN		(* Resets values *)
			(* uiSignalOutShared.00 & 01	--> X ekstra bits	: 00 --> +256 & 01 -->+512	*)
			(* uiSignalOutShared.02 & 03	--> Y ekstra bits	: 02 --> +256 & 03 -->+512	*)
			(* uiSignalOutShared.04 & 05	--> Z ekstra bits	: 04 --> +256 & 05 -->+512	*)

			(* G variablerne bliver sat i Control programmerne *)
			viX := GviX;						(*GviX - Global variable for Pos X *)
			viY := GviY;						(*GviY - Global variable for Pos Y *)
			viZ := GviZ;						(*GviZ - Global variable for Pos Z *)
			viA := GviA;						(*GviA - Global variable for Pos A *)
			viE := GviE;						(*GviE - Global variable for Pos E *)
			viR := GviR;						(*GviR - Global variable for Pos R *)

			(* ------------------------------ Negative Check ------------------------------ *)
			IF viX < 0 THEN							(* If X is negative, set orientation bit high *)
				uiSignalOutOrientation.03 := TRUE;
				viX := ABS(viX);
			ELSE
				uiSignalOutOrientation.03 := FALSE;
			END_IF
			IF viY < 0 THEN							(* If Y is negative, set orientation bit high *)
				uiSignalOutOrientation.04 := TRUE;
				viY := ABS(viY);
			ELSE
				uiSignalOutOrientation.04 := FALSE;
			END_IF
			IF viZ < 0 THEN							(* If Z is negative, set orientation bit high *)
				uiSignalOutOrientation.05 := TRUE;
				viZ := ABS(viZ);
			ELSE
				uiSignalOutOrientation.05 := FALSE;
			END_IF
			GsendCoord := FALSE;
			NewState := 10;
		END_IF

	10:		(* X Koordinat *)
		IF viX <> 0 THEN
			uiSignalOutShared.00 := FALSE;
			uiSignalOutShared.01 := FALSE;
			IF viX < 256 THEN
				(* Hvis koordinate er under 255 *)
				uiSignalOutX := INT_TO_BYTE(viX);
			ELSIF viX > 255 AND viX < 512THEN
				(* Hvis koordinat er mellem 255 og 511 *)
				uiSignalOutShared.00 := TRUE;
				uiSignalOutX := INT_TO_BYTE(viX  - 256);
			ELSE
				(* Hvis koordinat er over 512 *)
				IF viX - 512 > 255 THEN
					(* Hvis koordinat er over 768 skal begge ekstra bit vær høj*)
					uiSignalOutX := INT_TO_BYTE(viX  -  512 - 256);
					uiSignalOutShared.00 := TRUE;
					uiSignalOutShared.01 := TRUE;
				ELSE
					(* Hvis koordinat er mellem 512 og 767*)
					uiSignalOutX := INT_TO_BYTE(viX  -  512);
					uiSignalOutShared.01 := TRUE;
				END_IF
			END_IF
		END_IF
		NewState := 20;

	20:		(* Y Koordinat *)
		IF viY <> 0 THEN
			uiSignalOutShared.02 := FALSE;
			uiSignalOutShared.03 := FALSE;
			IF viY < 256 THEN
				(* Hvis koordinate er under 255 *)
				uiSignalOutY := INT_TO_BYTE(viY);
			ELSIF viY > 255 AND viY < 512THEN
				(* Hvis koordinat er mellem 255 og 511 *)
				uiSignalOutShared.02 := TRUE;
				uiSignalOutY := INT_TO_BYTE(viY  - 256);
			ELSE
				(* Hvis koordinat er over 512 *)
				IF viY - 512 > 255 THEN
					(* Hvis koordinat er over 768 skal begge ekstra bit vær høj*)
					uiSignalOutY := INT_TO_BYTE(viY  -  512 - 256);
					uiSignalOutShared.02 := TRUE;
					uiSignalOutShared.03 := TRUE;
				ELSE
					(* Hvis koordinat er mellem 512 og 767*)
					uiSignalOutY := INT_TO_BYTE(viY  -  512);
					uiSignalOutShared.03 := TRUE;
				END_IF
			END_IF
		END_IF
		NewState := 30;

	30:		(* Z Koordinat *)
		IF viZ <> 0 THEN
			uiSignalOutShared.04 := FALSE;
			uiSignalOutShared.05 := FALSE;
			IF viZ < 256 THEN
				(* Hvis koordinate er under 255 *)
				uiSignalOutZ := INT_TO_BYTE(viZ);
			ELSIF viZ > 255 AND viZ < 512THEN
				(* Hvis koordinat er mellem 255 og 511 *)
				uiSignalOutShared.04 := TRUE;
				uiSignalOutZ := INT_TO_BYTE(viZ  - 256);
			ELSE
				(* Hvis koordinat er over 512 *)
				IF viZ - 512 > 255 THEN
					(* Hvis koordinat er over 768 skal begge ekstra bit vær høj*)
					uiSignalOutZ := INT_TO_BYTE(viZ  -  512 - 256);
					uiSignalOutShared.04 := TRUE;
					uiSignalOutShared.05 := TRUE;
				ELSE
					(* Hvis koordinat er mellem 512 og 767*)
					uiSignalOutZ := INT_TO_BYTE(viZ  -  512);
					uiSignalOutShared.05 := TRUE;
				END_IF
			END_IF
		END_IF
		NewState := 40;

	40:		(* A Orientering *)
		(* Hvis negativ vinkel *)
		(* viA := viA / 100; *)
		IF viA < 0 THEN
			uiSignalOutA := INT_TO_BYTE(viA * -1);
			uiSignalOutOrientation.00 := TRUE;
		ELSE
			uiSignalOutA := INT_TO_BYTE(viA);
			uiSignalOutOrientation.00 := FALSE;
		END_IF

		NewState := 50;

	50:
		(* Hvis negativ vinkel *)
		(* viE := viE / 100; *)
		IF viE < 0 THEN
			uiSignalOutE := INT_TO_BYTE(viE * -1);
			uiSignalOutOrientation.01 := TRUE;
		ELSE
			uiSignalOutE := INT_TO_BYTE(viE);
			uiSignalOutOrientation.01 := FALSE;
		END_IF
		NewState := 60;

	60:
		(* Hvis negativ vinkel*)
		(* viR := viR / 100; *)
		IF viR < 0 THEN
			uiSignalOutR := INT_TO_BYTE(viR * -1);
			uiSignalOutOrientation.02 := TRUE;
		ELSE
			uiSignalOutR := INT_TO_BYTE(viR);
			uiSignalOutOrientation.02 := FALSE;
		END_IF

		NewState := 70;

	70:		(* Pick angle *)
		(* Hvis negativ vinkel*)
		(* viR := viR / 100; *)
		IF GviPick < 0 THEN
			uiSignalOutPick := INT_TO_BYTE(ABS(GviPick));
			uiSignalOutOrientation.06 := TRUE;
		ELSE
			uiSignalOutPick := INT_TO_BYTE(GviPick);
			uiSignalOutOrientation.06 := FALSE;
		END_IF

		NewState := 80;

	80:		(* X2  *)
		(* Hvis negativ *)
		IF GviX2 < 0 THEN
			uiSignalOutX2 := ABS(GviX2);
		ELSE
			uiSignalOutX2 := GviX2;
		END_IF

		NewState := 90;

	90:		(* Y2  *)
		(* Hvis negativ *)
		IF GviY2 < 0 THEN
			uiSignalOutY2 := ABS(GviY2);
		ELSE
			uiSignalOutY2 := GviY2;
		END_IF

		NewState := 100;

	100:		(* Z2  *)
		(* Hvis negativ *)
		IF GviZ2 < 0 THEN
			uiSignalOutZ2 := ABS(GviZ2);
		ELSE
			uiSignalOutZ2 := GviZ2;
		END_IF

		NewState := 1000;


	1000:		(* Reset global variable Pos efter robot Cut har modtaget den *)
		uiSignalOutShared.06 := TRUE;			(* Acknowledge that Pos is sent *)
		GcoordSent := TRUE;
		GsendCoord := FALSE;
		(* IF the position has been recieved and maybe sent to Pick --> Reset variables *)
		IF uiSignalIn4.00 THEN
			uiSignalOutShared.06 := FALSE;		(* Pos sent Acknowledge *)
			GviX := 0;
			GviY := 0;
			GviZ := 0;
			GviA := 0;
			GviE := 0;
			GviR := 0;
			NewState := 0;
		END_IF

END_CASE

END_PROGRAM

// ---- POUs/PcCom.TcPOU
PROGRAM PcCom
VAR_INPUT
	State: INT := 0;
END_VAR


VAR

	NewState: INT := 0;


	byTest : ARRAY[0..1]OF BYTE;
	nTest : UINT;

	setToNull: BOOL;

	bCut: BOOL;
	Wait: TON;
	bWait: BOOL;
	CollectImages: BOOL;
	bWait1: BOOL;
	Wait1: TON;
	CutCam: BOOL;
	PickCam: BOOL;
	imgCount: INT;
END_VAR
VAR_OUTPUT
	bPick: BOOL;
END_VAR

(* Til at sende og modtage data Mellem PLC og PC *)

CASE State OF


0: (*INIT*)
(*Output*)

	(* Reset data sent to PC *)
	stDataToVision.CmdByte		:= 0;
	stDataToVision.CmdIdOut		:= 0;
	stDataToVision.ResultRead	:= 0;
	stDataToVision.CoordXR1G	:= 0;
	stDataToVision.CoordYR1G	:= 0;
	stDataToVision.CoordZR1G	:= 0;
	stDataToVision.CoordXR2G	:= 0;
	stDataToVision.CoordYR2G	:= 0;
	stDataToVision.CoordZR2G	:= 0;
	stDataToVision.CoordRRA		:= 0;
	stDataToVision.CoordRRE		:= 0;
	stDataToVision.CoordRRR		:= 0;

	gResetPcCom 	:= FALSE;
	NewState 		:= 10;

10:
		(*	------------------------------Cut position------------------------------	*)
		(* If Cut pos needs to be sent to PC *)
		IF getCutCoords  AND NOT getPickCoords THEN
			FB_GET_CUT_COORD.Execute := TRUE;
			uiSignalOutControl := FB_GET_CUT_COORD.OutQ;		(* Retreives Pick pos from robotPick *)
			IF FB_GET_CUT_COORD.Done THEN	(* Check for pos sent. When acknowledge the pos is sent to PLC *)
				FB_GET_CUT_COORD.Execute := FALSE;
				GgetCoord := TRUE;						(* Starts GetCoordinates *)
				getCutCoords := FALSE;
			END_IF
		END_IF

		(*	------------------------------Pick position------------------------------	*)
		IF getPickCoords  AND NOT getCutCoords THEN
			FB_GET_PICK_COORD.Execute := TRUE;
			uiSignalOutControl := FB_GET_PICK_COORD.OutQ;		(* Retreives Pick pos from robotPick *)
			IF FB_GET_PICK_COORD.Done THEN	(* Check for pos sent. When acknowledge the pos is sent to PLC *)
				FB_GET_PICK_COORD.Execute := FALSE;
				GgetCoord := TRUE;						(* Starts GetCoordinates *)
				getPickCoords := FALSE;
			END_IF
		END_IF

		IF CutCoord THEN									(* If coordinates from cut has sbeen recieved, send to PC *)
			(* CoordRG	--> Mapped to fieldbus Com to PC *)
			stDataToVision.CoordXR1G := currentRobotX;
			stDataToVision.CoordYR1G := currentRobotY;
			stDataToVision.CoordZR1G := currentRobotZ;
			stDataToVision.CoordRRA:= currentRobotA;
			stDataToVision.CoordRRE := currentRobotE;
			stDataToVision.CoordRRR := currentRobotR;
			bPosSentToPcCom := TRUE;
			CutCoord := FALSE;
		END_IF

		IF PickCoord THEN								(* If coordinates from pick has sbeen recieved, send to PC *)
			(* CoordRG	--> Mapped to fieldbus Com to PC *)
			stDataToVision.CoordXR2G := currentRobotX;
			stDataToVision.CoordYR2G := currentRobotY;
			stDataToVision.CoordZR2G := currentRobotZ;
			stDataToVision.CoordRRA:= currentRobotA;
			stDataToVision.CoordRRE := currentRobotE;
			stDataToVision.CoordRRR := currentRobotR;
			bPosSentToPcCom := TRUE;
			FB_GET_PICK_COORD.Execute := FALSE;
			PickCoord := FALSE;
		END_IF

		IF gResetPcCom THEN
			NewState := 0;
		END_IF

END_CASE

(* When PC has read the Command *)
IF stDataToVision.ResultRead = 1 THEN
	stDataToVision.CmdByte := 0;
END_IF

(* HMI bottons for controlling PC *)
IF bHelloWorld THEN
	stDataToVision.CmdByte := 1;
ELSIF bCalibCamOneStart THEN
	stDataToVision.CmdByte := 2;
ELSIF bNewPosCalibCamOne THEN
	stDataToVision.CmdByte := 3;
ELSIF bEndCalibCamOne THEN
	stDataToVision.CmdByte := 4;
ELSIF bCalibCamTwoStart THEN
	stDataToVision.CmdByte := 5;
ELSIF bNewPosCalibCamTwo THEN
	stDataToVision.CmdByte := 6;
ELSIF bEndCalibCamTwo THEN
	stDataToVision.CmdByte := 7;
ELSIF bStartStopPlantCheck THEN
	stDataToVision.CmdByte := 8;
ELSIF bStopCheck THEN
	stDataToVision.CmdByte := 9;
ELSIF bGetPlantDataCamOne THEN
	stDataToVision.CmdByte := 10;
ELSIF bGetPlantDataCamTwo THEN
	stDataToVision.CmdByte := 12;
ELSIF bRestart THEN
	stDataToVision.CmdByte := 14;
ELSIF bShutdown THEN
	stDataToVision.CmdByte := 15;
ELSIF bTestCamPointCam2 THEN
	stDataToVision.CmdByte := 13;
ELSIF bTestCamPointCam1 THEN
	stDataToVision.CmdByte := 11;
ELSIF usiVisionCmd <> 0 THEN
	stDataToVision.CmdByte := usiVisionCmd;
ELSIF usiVisionCmd = 0 THEN
	stDataToVision.CmdByte := 0;
END_IF

IF CollectImages THEN
	IF stDataToVision.CmdByte = 0 AND NOT bGetPlantDataCamOne AND NOT bGetPlantDataCamTwo AND Wait1.Q THEN
		IF CutCam THEN
			bGetPlantDataCamOne := TRUE;
		ELSIF PickCam THEN
			bGetPlantDataCamTwo := TRUE;
		END_IF
		bWait := TRUE;
		bWait1 := FALSE;
	END_IF
	
	IF Wait.Q THEN
		bWait1 := TRUE;
		bWait := FALSE;
		imgCount := imgCount + 1;
		bGetPlantDataCamOne := FALSE;
		bGetPlantDataCamTwo := FALSE;
	END_IF
END_IF

FB_CAM_ONE_CONTROL(ControlType := 1,			Command => bTestCamPointCam1,	CommandNo := stDataFromVision.CmdInProcess, 	Ack := stDataToVision.CmdByte, 	TrunkPosY := stDataFromVision.ResultPar2,
							BunchPosX := stDataFromVision.ResultPar4,		BunchPosY := stDataFromVision.ResultPar5,		BunchPosZ := stDataFromVision.ResultPar6,		StemAngle := stDataFromVision.ResultPar7);
FB_CAM_TWO_CONTROL(ControlType := 1,			Command => bTestCamPointCam2,	CommandNo := stDataFromVision.CmdInProcess,	Ack := stDataToVision.CmdByte,	X := stDataFromVision.ResultPar1, 	Y := stDataFromVision.ResultPar2, 	Z := stDataFromVision.ResultPar3,
							RotZ0 := stDataFromVision.ResultPar4,	RotY := stDataFromVision.ResultPar5,	RotZ1 := stDataFromVision.ResultPar6, StemHeading := stDataFromVision.ResultPar7,	StemFound :=stDataFromVision.gStemFound, JointFound := stDataFromVision.gJointFound,
							TomatoFound := stDataFromVision.gTomatoFound, TrussFound := stDataFromVision.gTrussFound);
							
Wait			(IN:=  bWait			, PT:=T#500MS, Q=>, ET=>);
Wait1			(IN:=  bWait1			, PT:=T#500MS, Q=>, ET=>);

END_PROGRAM

// ---- POUs/ErrorHandle.TcPOU
PROGRAM ErrorHandle
VAR_INPUT
	State: INT := 0;
END_VAR

VAR

	uiSignalOutAlarm : BYTE;
	uiSignalInAlarmCode : UDINT;
	uiSignalInAlarm : BYTE;

	NewState: INT := 0;

	bCancelAlarm: BOOL;
	bPickRobot: BOOL;
	bCutRobot: BOOL;
	bErrorWhere: INT;

	sSeverity: STRING;
	iLen: INT;
	iSeverity: USINT;

	(*Timer*)
	TonWait : TON;

	ilentemp: INT;
	sString: STRING(255);
	updateFlag: BOOL;
END_VAR

CASE State OF

	0:		(* Kig efter om der er opstået en fejl *)
		IF uiSignalInAlarmCode <> 0 THEN
			robotAlarmId := uiSignalInAlarmCode;
			(* Hvis der er en fejl, sat HMI i alarm state *)
			bAlarmState := TRUE;
			(* Find ud af hvilken robot der kommer med fejlen *)
			IF bErrorWhere = 1 THEN
				sDeviceWhich := 'Robot Cut';
				bCutRobot := TRUE;
			ELSIF bErrorWhere = 2 THEN
				sDeviceWhich := 'Robot Pick';
				bPickRobot := TRUE;
			END_IF
			NewState := 10;
		END_IF
		
	10:		(* Look in DB for alarm severity *)
		P_SqlSelectAlarm.bRead := TRUE;
		IF P_SqlSelectAlarm.bDone THEN
			P_SqlSelectAlarm.bRead := FALSE;
			
			// Get alarm description and find severity
			sString		:= RIGHT(P_SqlSelectAlarm.astData[0].alarmDesc, LEN(P_SqlSelectAlarm.astData[0].alarmDesc) - 1);
			iLen 		:= FIND(sString, '-');
			ilentemp := iLen;
			sSeverity 	:= LEFT( P_SqlSelectAlarm.astData[0].alarmDesc, iLen);
			iSeverity 	:= TO_USINT(sSeverity);
			IF iSeverity >= 4 THEN
				bStop := TRUE;
				NewState := 20;
			ELSE
				NewState := 30; //30
			END_IF
		END_IF
		
	20:		(* Send alarm ID to MQTT broker *)
		(* Stop running - Virker endnu ikke *)
		gSeverity := iSeverity;
		uiSignalOut3.00 := TRUE;
		bNoDriveOff := FALSE;
		bAlarm := TRUE;
		NewState := 30;
	
		
	30:		(* Input alarm in DB table alarmLog *)
		IF (sDeviceWhich <> '') THEN
			P_SqlInsertAlarmLog.bInsert := TRUE;
			IF P_SqlInsertAlarmLog.bDone THEN
				P_SqlInsertAlarmLog.bInsert := FALSE;
				NewState := 40;
			END_IF
		ELSE
			robotAlarmId := 999; // Unknown PLC error
			sDeviceWhich := 'PLC';
			P_SqlInsertAlarmLog.bInsert := TRUE;
			IF P_SqlInsertAlarmLog.bDone THEN
				P_SqlInsertAlarmLog.bInsert := FALSE;
				NewState := 40;
			END_IF
		END_IF
		
	40:		(* Wait for alarm to be acknowledged *)
		IF NOT bAlarm THEN
			sDeviceWhich := '';
			robotAlarmId := 0;
			bAlarmAck := TRUE;
			NewState := 50;
		END_IF
		
	50:		(* Reset, og gør klar til at køre igen *)
		bAlarmAck := FALSE;
		uiSignalOut3.00 := FALSE;
		bNoDriveOff := TRUE;
		bCancelAlarm := TRUE;
		TonWait.IN := TRUE;
		IF TonWait.Q THEN
			TonWait.IN := FALSE;
			bCancelAlarm := FALSE;
			uiAlarm := 0;
			gSeverity := 0; 
			bAlarmState := FALSE;
			uiStatus := 0;
			NewState  := 0;
		END_IF

END_CASE

bErrorWhere := WhichRobot;
uiSignalInAlarmCode := ErrorNum;
uiAlarm := uiSignalInAlarmCode;
CancelAlarm := BOOL_TO_BYTE(bCancelAlarm);

(*
bErrorWhere := uiSignalInAlarm;
uiAlarm := uiSignalInAlarmCode;
uiSignalOutAlarm.00 := bCancelAlarm;*)

IF uiSignalInAlarmCode = 0  AND NewState = 10 THEN
	bAckAlarm := FALSE;
END_IF

TonWait(IN:=State = 50,	PT:=t#1000ms ,	Q=> ,	ET=> );

END_PROGRAM

// ---- POUs/GetCoordinates.TcPOU
 PROGRAM GetCoordinates
VAR_INPUT
	State: INT :=0;
END_VAR

VAR

	NewState: INT := 0;

	Wait: TON;
	bWait: BOOL;
END_VAR

(* For getting robot coordinates *)

CASE State OF

	0:
		bReady := TRUE;
		IF GgetCoord THEN		(* Start reading Robot Pos *)
			bReady := FALSE;
			GgetCoord := FALSE;
			bGetCoordDone := FALSE;
			CutCoord := FALSE;	(* Blev sat HIGH, da en forspørges på pick koordinat var ønsket *)
			PickCoord := FALSE;	(* Blev sat HIGH, da en forspørges på cut koordinat var ønsket *)
			NewState := 10;
		END_IF

	10:		(* X Koordinat - Unwrapping the positions *)
		currentRobotX := uiSignalInX;
		IF uiSignalInOrientation.03 THEN
			currentRobotX := currentRobotX * -1;
		END_IF
		NewState := 20;

	20:		(* Y Koordinat - Unwrapping the positions *)
		currentRobotY := uiSignalInY;
		IF uiSignalInOrientation.04 THEN
			currentRobotY := currentRobotY * -1;
		END_IF
		NewState := 30;

	30:		(* Z Koordinat - Unwrapping the positions *)
		currentRobotZ := uiSignalInZ;
		IF uiSignalInOrientation.05 THEN
			currentRobotZ := currentRobotZ * -1;
		END_IF
		NewState := 40;

	40:		(* A Orientering - Her er det ikke nødvendigt at pakke ud, da der bliver brugt 16 bits til at sende rotation. Derfor værdier op til 65.535*)
		(* Hvis negativ vinkel *)
		IF uiSignalInOrientation.00 THEN
			currentRobotA := uiSignalInA * -1;
		ELSE
			currentRobotA := uiSignalInA;
		END_IF

		NewState := 50;

	50:
		(* Hvis negativ vinkel - Her er det ikke nødvendigt at pakke ud, da der bliver brugt 16 bits til at sende rotation. Derfor værdier op til 65.535 *)
		IF uiSignalInOrientation.01 THEN
			currentRobotE := uiSignalInE * -1;
		ELSE
			currentRobotE := uiSignalInE;
		END_IF

		NewState := 60;

	60:
		(* Hvis negativ vinkel - Her er det ikke nødvendigt at pakke ud, da der bliver brugt 16 bits til at sende rotation. Derfor værdier op til 65.535*)
		IF uiSignalInOrientation.02 THEN
			currentRobotR := uiSignalInR * -1;
		ELSE
			currentRobotR := uiSignalInR;
		END_IF

		NewState := 70;

	70:		(* Hvis uiSignalInShared.06 er HIGH, er det koordinater fra Cut der bliver sendt. Ellers er det Pick *)
			(* Sends to PcCom *)
			IF uiSignalInShared.06 THEN
				CutCoord := TRUE;
				PickCoord := FALSE;
			END_IF
			IF NOT uiSignalInShared.06 THEN
				CutCoord := FALSE;
				PickCoord := TRUE;
			END_IF
			bGetCoordDone := TRUE;
			bGetCutCoordDone:= TRUE;
			NewState := 0;


END_CASE

Wait		(IN:=  bWait		, PT:=t#400ms, Q=>, ET=>); 	(*Timer*)

END_PROGRAM

// ---- POUs/CONTROLs/CalibCam1.TcPOU
PROGRAM CalibCam1
VAR_INPUT
	State: INT :=0;
	NewState: INT := 0;
	next: BOOL;
END_VAR

VAR
	bCommandStarted: BOOL;

	Wait: TON;
	bWait: BOOL;
	Wait2: TON;
	bWait2: BOOL;
	Wait3: TON;
	bWait3: BOOL;
	bStopped: BOOL;
END_VAR

IF sNewCalib = 'he-cut-start' THEN
	startCalibCam1 := TRUE;
ELSE
	startCalibCam1 := FALSE;
END_IF

CASE State OF

	0:		(* Wait for start of Calib cam 1 *)
		IF (uiprogNo = 1 OR allZero) AND startCalibCam1 AND State <> 2000  AND NOT bAlarmState THEN
			uiCalibImgCount := 0;
			uiSignalOutTool.06 := TRUE;
			startCalibCam1 := FALSE;
			GbCloseCut := TRUE;									(* When calibrating Cam 1, the cutter most be closed *)
			NewState := 10;
		END_IF

	10:		(* Set calibration velocity *)
		uiSignalOutSpeedControl := UINT_TO_BYTE(uiSpeedSetting);
		uiSignalOutControl := Set_Velocity;

		IF uiSignalInAck = Set_Velocity THEN
			uiSignalOutControl := 0;
			NewState := 15;
		END_IF

	15:
		IF uiSignalInAck = 0 THEN
			NewState := 20;
		END_IF

